REGION Network 6: Выходной сигнал контроллера
   RUNG wire#powerrail
      Contact( #CMD.Start_M )
      Move(in := 1, out1 => #Status)
      I_Contact( #Use.Inverse )
      wire#w1
      I_Contact( #All_Block )
      I_Contact( "Sim_All" )
      I_Contact( #CMD.Sim )
      I_Contact( #CMD.Local )
      Coil( #Q )
   END_RUNG
   RUNG wire#powerrail
      I_Contact( #CMD.Start_M )
      Move(in := 0, out1 => #Status)
      Contact( #Use.Inverse )
   END_RUNG wire#w1
   // the same network as SCL:
   IF #CMD.Start_M THEN #Status := 1; END_IF;
   IF NOT #CMD.Start_M THEN #Status := 0; END_IF;
   #Q := ((#CMD.Start_M AND NOT #Use.Inverse) OR (NOT #CMD.Start_M AND #Use.Inverse)) AND NOT #All_Block AND NOT "Sim_All" AND NOT #CMD.Sim AND NOT #CMD.Local;
END_REGION

REGION Network 7: Косвенная адресация
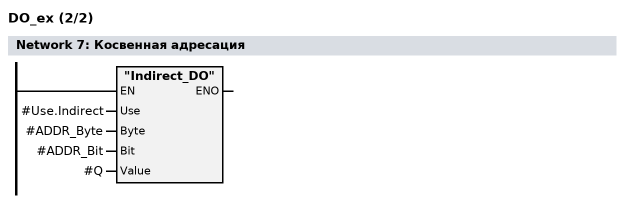
   RUNG wire#powerrail
      "Indirect_DO"(Use := #Use.Indirect, "Byte" := #ADDR_Byte, Bit := #ADDR_Bit, Value := #Q)
   END_RUNG
   // the same network as SCL:
   "Indirect_DO"(Use := #Use.Indirect, "Byte" := #ADDR_Byte, Bit := #ADDR_Bit, Value := #Q);
END_REGION
END_FUNCTION_BLOCK

FUNCTION_BLOCK "Motors"   // FB240, LAD
{ S7_Optimized_Access := 'FALSE' }
VERSION : 0.1
// stored: AutoNumber false, IsIECCheckEnabled false, SetENOAutomatically false, UDAEnableTagReadback false
   VAR DB_SPECIFIC
      Time_DTL { S7_SetPoint := 'True'} : DTL;
   END_VAR
BEGIN

REGION Network 1: Мешалки
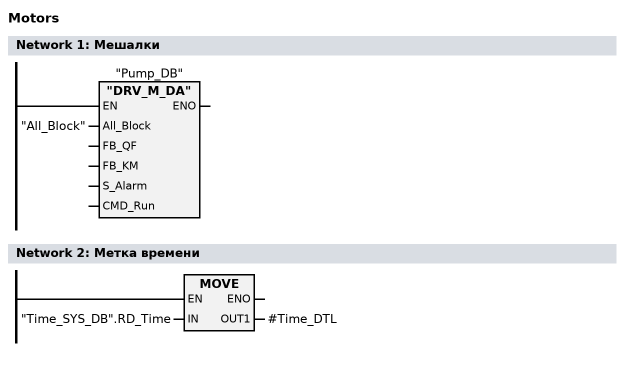
   RUNG wire#powerrail
      "Pump_DB"(All_Block := "All_Block", FB_QF :=, FB_KM :=, S_Alarm :=, CMD_Run :=)
   END_RUNG
   // the same network as SCL:
   "Pump_DB"(All_Block := "All_Block");   // "DRV_M_DA"
END_REGION

REGION Network 2: Метка времени
   RUNG wire#powerrail
      Move(in := "Time_SYS_DB".RD_Time, out1 => #Time_DTL)
   END_RUNG
   // the same network as SCL:
   #Time_DTL := "Time_SYS_DB".RD_Time;
END_REGION
END_FUNCTION_BLOCK

FUNCTION_BLOCK "DRV_M_DA"   // FB111, LAD
{ S7_Optimized_Access := 'FALSE' }
VERSION : 0.1
// stored: AutoNumber false, IsIECCheckEnabled false, SetENOAutomatically false, UDAEnableTagReadback false
   VAR_INPUT
      All_Block : Bool;   // Аварийный останов
   END_VAR
   VAR_IN_OUT
      FB_QF : Bool;   // защитный автомат / Защитный автомат / Готовность
      FB_KM : Bool;   // привод запущен / Пускатель / В работе
      S_Alarm : Bool;   // Внешний индикатор наличия аварии
      CMD_Run : Bool;   // Команда запуска двигателя
   END_VAR
   VAR DB_SPECIFIC
      CMD : "CMD";   // Основные команды / Блок команд
      Mode : Int;   // Режим работы
      Status : Int;   // Статус устройства
      Use : Struct   // Функционал
         QF { S7_SetPoint := 'True'} : Bool := true;   // Защитный автомат
         KM { S7_SetPoint := 'True'} : Bool := true;   // Пускатель
         OpTime { S7_SetPoint := 'True'} : Bool := true;   // Контроль наработки
         Analog { S7_SetPoint := 'True'} : Bool := true;
         Local_Keys : Bool;
      END_STRUCT;
      FB : Struct   // Функционал
         QF : Bool;   // Защитный автомат
         KM : Bool;   // Пускатель
         Local_Start : Bool;
         Local_Stop : Bool;
      END_STRUCT;
      ON : Bool;   // Успешно запущено
      OFF : Bool;   // Успешно остановлено
   END_VAR
   VAR
      Tx { S7_SetPoint := 'True'} : Array[0..3] of "Time_S";   // Блок таймеров
   END_VAR
   VAR DB_SPECIFIC
      Inv : Struct   // Инверсия сигналов
         CMD { S7_SetPoint := 'True'} : Bool;   // Команда запуска
         QF { S7_SetPoint := 'True'} : Bool;   // Защитный автомат
         KM { S7_SetPoint := 'True'} : Bool;   // Пускатель
      END_STRUCT;
      Alarm : Struct   // Сбор аварий / Список аварий
         Block : Bool;   // Аварийная остановка
         QF : Bool;   // привод не готов / Выбило защитный автомат
         Start : Bool;   // Ошибка при запуске
         Stop : Bool;   // Ошибка при останове
         Termo : Bool;   // термозащита / Сработала термозащита
         Alarm : Bool;   // Внешняя авария
         Safety : Bool;   // Сработала безопасность
         OpTime : Bool;
      END_STRUCT;
      Alarms : Word;   // Слово аварий
      Events : Word;   // События
      pos : Array[0..15] of Bool;
      OpTime_h : DInt;   // наработка (ч)
      OpTime_s { S7_SetPoint := 'True'} : DInt;   // наработка (с)
      OpTime_SP { S7_SetPoint := 'True'} : DInt := 2160;   // Интервал обслуживания, ч
      OpTime_Now_h : DInt;   // Прошло с прошлого обслуживания, ч
      OpTime_Now_s { S7_SetPoint := 'True'} : DInt;   // Прошло с прошлого обслуживания, с
      CodeID { S7_SetPoint := 'True'} : Int;   // Код датчика для привязки в скаде
      Indirect : Struct   // Использование косвенной адресации
         FB_QF { S7_SetPoint := 'True'} : Bool := true;   // защитный автомат / Защитный автомат
         FB_KM { S7_SetPoint := 'True'} : Bool := true;   // привод запущен / Пускатель
         CMD { S7_SetPoint := 'True'} : Bool := true;   // Команда запуска привода
      END_STRUCT;
      Indirect_BYTE : Struct   // Адрес входа на контроллере (Байт)
         FB_QF { S7_SetPoint := 'True'} : Int;   // защитный автомат / Защитный автомат
         FB_KM { S7_SetPoint := 'True'} : Int;   // привод запущен / Пускатель
         CMD { S7_SetPoint := 'True'} : Int;   // Команда запуска привода
      END_STRUCT;
      Indirect_BIT : Struct   // Адрес входа на контроллере (Бит)
         FB_QF { S7_SetPoint := 'True'} : Int := 9;   // защитный автомат / Защитный автомат
         FB_KM { S7_SetPoint := 'True'} : Int := 9;   // привод запущен / Пускатель
         CMD { S7_SetPoint := 'True'} : Int := 9;   // Команда запуска привода
      END_STRUCT;
      SP_A : Real;   // Уставка скорости в авторежиме
      SP_M : Real;   // Уставка скорости в ручном режиме
      ADDR { S7_SetPoint := 'True'} : Int;   // Уставка
   END_VAR
   VAR
      Converter { S7_SetPoint := 'True'} : "Converter_SCL";   // Масштабирование сигнала
   END_VAR
   VAR DB_SPECIFIC
      VmA : Real;   // Реальный сигнал на входе ПЛК
      Output_Type { S7_SetPoint := 'True'} : Int;   // Тип выхода, 0 - 4..20, 1 - 0..20, 2 - 0..10, 3 - 0..5
      "Type" { S7_SetPoint := 'True'} : Int;   // Размерность
   END_VAR
   VAR
      Slow { S7_SetPoint := 'True'} : "Slow";   // Плавный разгон и замедление
   END_VAR
   VAR DB_SPECIFIC
      "Name" { S7_SetPoint := 'True'} : String[4];
      coeff : Real;
      SP_Min { S7_SetPoint := 'True'} : Real := 30.0;
      Time_DTL { S7_SetPoint := 'True'} : DTL;
   END_VAR
   VAR_TEMP
      ev : Bool;
      xQF : Bool;
      xKM : Bool;
      xSP : Real;
      Signal_R : Real;   // Актуальный сигнал
      Signal_Dint : DInt;   // Сигнал в DInt
      Signal_Ex : Int;   // Конвертация сигнала
      Type_Min : Real;
      Type_Max : Real;
   END_VAR
   // Converter.Max_In := 100.0;
   // Converter.Max_Out := 27648.0;
   VAR_TEMP   // added for the SCL form of the ladder/FBD networks
      _w1 : Bool;
      _w2 : Bool;
      _w3 : Bool;
      _w4 : Bool;
      _w5 : Bool;
      _w6 : Bool;
      _w7 : Bool;
      _w8 : Bool;
      _w9 : Bool;
      _w10 : Bool;
      _w11 : Bool;
      _w12 : Bool;
      _w13 : Bool;
      _w14 : Bool;
      _w15 : Bool;
      _w16 : Bool;
      _w17 : Bool;
      _w18 : Bool;
      _w19 : Bool;
      _w20 : Bool;
      _w21 : Bool;
      _w22 : Bool;
      _w23 : Bool;
      _w24 : Bool;
      _w25 : Bool;
      _w26 : Bool;
   END_VAR
BEGIN

REGION Network 1: Режим глобальной симуляции
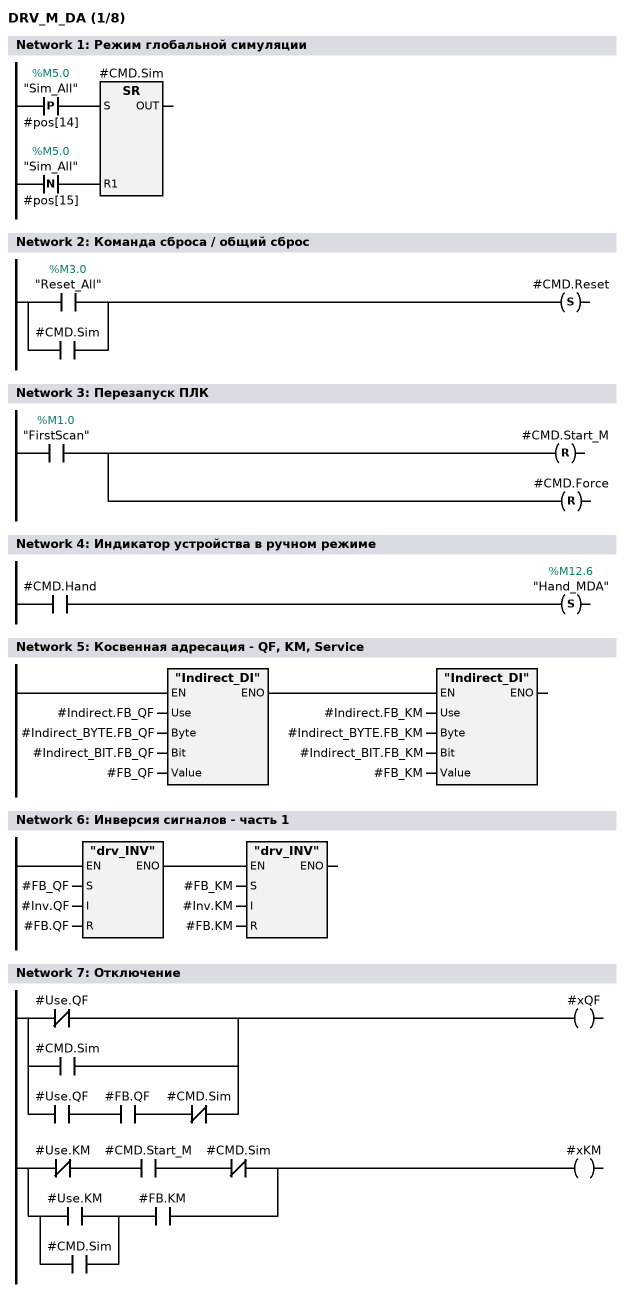
   RUNG wire#powerrail
      P_Contact(operand := "Sim_All", bit := #pos[14])
      S_SR(operand := #CMD.Sim, r1 := wire#w1)
   END_RUNG
   RUNG wire#powerrail
      N_Contact(operand := "Sim_All", bit := #pos[15])
   END_RUNG wire#w1
   // the same network as SCL:
   #_w1 := "Sim_All" AND NOT #pos[14];   // rising edge of "Sim_All"
   #pos[14] := "Sim_All";
   #_w2 := NOT "Sim_All" AND #pos[15];   // falling edge of "Sim_All"
   #pos[15] := "Sim_All";
   IF #_w1 THEN
       #CMD.Sim := TRUE;   // SR flip-flop
   END_IF;
   IF #_w2 THEN #CMD.Sim := FALSE; END_IF;
END_REGION

REGION Network 2: Команда сброса / общий сброс
   RUNG wire#powerrail
      Contact( "Reset_All" )
      wire#w1
      S_Coil( #CMD.Reset )
   END_RUNG
   RUNG wire#powerrail
      Contact( #CMD.Sim )
   END_RUNG wire#w1
   // the same network as SCL:
   IF "Reset_All" OR #CMD.Sim THEN #CMD.Reset := TRUE; END_IF;
END_REGION

REGION Network 3: Перезапуск ПЛК
   RUNG wire#powerrail
      Contact( "FirstScan" )
      wire#w1
      R_Coil( #CMD.Start_M )
   END_RUNG
   RUNG wire#w1
      R_Coil( #CMD.Force )
   END_RUNG
   // the same network as SCL:
   IF "FirstScan" THEN
       #CMD.Start_M := FALSE;
       #CMD.Force := FALSE;
   END_IF;
END_REGION

REGION Network 4: Индикатор устройства в ручном режиме
   RUNG wire#powerrail
      Contact( #CMD.Hand )
      S_Coil( "Hand_MDA" )
   END_RUNG
   // the same network as SCL:
   IF #CMD.Hand THEN "Hand_MDA" := TRUE; END_IF;
END_REGION

REGION Network 5: Косвенная адресация - QF, KM, Service
   RUNG wire#powerrail
      "Indirect_DI"(Use := #Indirect.FB_QF, "Byte" := #Indirect_BYTE.FB_QF, Bit := #Indirect_BIT.FB_QF, Value := #FB_QF)
      "Indirect_DI"(Use := #Indirect.FB_KM, "Byte" := #Indirect_BYTE.FB_KM, Bit := #Indirect_BIT.FB_KM, Value := #FB_KM)
   END_RUNG
   // the same network as SCL:
   "Indirect_DI"(Use := #Indirect.FB_QF,
                 "Byte" := #Indirect_BYTE.FB_QF,
                 Bit := #Indirect_BIT.FB_QF,
                 Value := #FB_QF,
                 ENO => #_w1);
   IF #_w1 THEN
       "Indirect_DI"(Use := #Indirect.FB_KM,
                     "Byte" := #Indirect_BYTE.FB_KM,
                     Bit := #Indirect_BIT.FB_KM,
                     Value := #FB_KM);
   END_IF;
END_REGION

REGION Network 6: Инверсия сигналов - часть 1
   RUNG wire#powerrail
      "drv_INV"(S := #FB_QF, I := #Inv.QF, R := #FB.QF)
      "drv_INV"(S := #FB_KM, I := #Inv.KM, R := #FB.KM)
   END_RUNG
   // the same network as SCL:
   "drv_INV"(S := #FB_QF, I := #Inv.QF, R := #FB.QF, ENO => #_w1);
   IF #_w1 THEN "drv_INV"(S := #FB_KM, I := #Inv.KM, R := #FB.KM); END_IF;
END_REGION

REGION Network 7: Отключение
   RUNG wire#powerrail
      I_Contact( #Use.QF )
      wire#w1
      Coil( #xQF )
   END_RUNG
   RUNG wire#powerrail
      Contact( #CMD.Sim )
   END_RUNG wire#w1
   RUNG wire#powerrail
      Contact( #Use.QF )
      Contact( #FB.QF )
      I_Contact( #CMD.Sim )
   END_RUNG wire#w1
   RUNG wire#powerrail
      I_Contact( #Use.KM )
      Contact( #CMD.Start_M )
      I_Contact( #CMD.Sim )
      wire#w2
      Coil( #xKM )
   END_RUNG
   RUNG wire#powerrail
      Contact( #Use.KM )
      wire#w3
      Contact( #FB.KM )
   END_RUNG wire#w2
   RUNG wire#powerrail
      Contact( #CMD.Sim )
   END_RUNG wire#w3
   // the same network as SCL:
   #xQF := NOT #Use.QF OR #CMD.Sim OR (#Use.QF AND #FB.QF AND NOT #CMD.Sim);
   #xKM := (NOT #Use.KM AND #CMD.Start_M AND NOT #CMD.Sim) OR ((#Use.KM OR #CMD.Sim) AND #FB.KM);
END_REGION

REGION Network 8: Режим работы устройства / определение режима работы
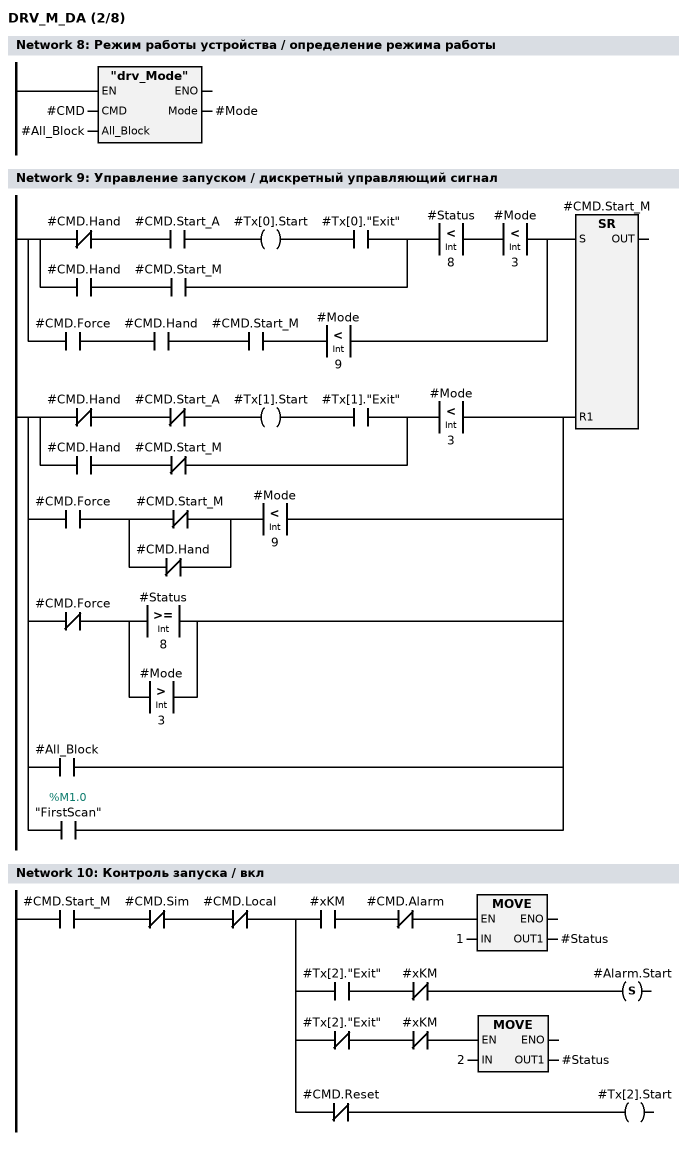
   RUNG wire#powerrail
      "drv_Mode"(CMD := #CMD, All_Block := #All_Block, Mode => #Mode)
   END_RUNG
   // the same network as SCL:
   "drv_Mode"(CMD := #CMD, All_Block := #All_Block, Mode => #Mode);
END_REGION

REGION Network 9: Управление запуском / дискретный управляющий сигнал
   RUNG wire#powerrail
      I_Contact( #CMD.Hand )
      Contact( #CMD.Start_A )
      Coil( #Tx[0].Start )
      Contact( #Tx[0]."Exit" )
      wire#w1
      { S7_Templates := "SrcType := Int" } LT_Contact(in1 := #Status, in2 := 8)
      { S7_Templates := "SrcType := Int" } LT_Contact(in1 := #Mode, in2 := 3)
      wire#w2
      S_SR(operand := #CMD.Start_M, r1 := wire#w7)
   END_RUNG
   RUNG wire#powerrail
      Contact( #CMD.Hand )
      Contact( #CMD.Start_M )
   END_RUNG wire#w1
   RUNG wire#powerrail
      Contact( #CMD.Force )
      Contact( #CMD.Hand )
      Contact( #CMD.Start_M )
      { S7_Templates := "SrcType := Int" } LT_Contact(in1 := #Mode, in2 := 9)
   END_RUNG wire#w2
   RUNG wire#powerrail
      I_Contact( #CMD.Hand )
      I_Contact( #CMD.Start_A )
      Coil( #Tx[1].Start )
      Contact( #Tx[1]."Exit" )
      wire#w3
      { S7_Templates := "SrcType := Int" } LT_Contact(in1 := #Mode, in2 := 3)
   END_RUNG wire#w7
   RUNG wire#powerrail
      Contact( #CMD.Hand )
      I_Contact( #CMD.Start_M )
   END_RUNG wire#w3
   RUNG wire#powerrail
      Contact( #CMD.Force )
      wire#w4
      I_Contact( #CMD.Start_M )
      wire#w5
      { S7_Templates := "SrcType := Int" } LT_Contact(in1 := #Mode, in2 := 9)
   END_RUNG wire#w7
   RUNG wire#w4
      I_Contact( #CMD.Hand )
   END_RUNG wire#w5
   RUNG wire#powerrail
      I_Contact( #CMD.Force )
      wire#w6
      { S7_Templates := "SrcType := Int" } GE_Contact(in1 := #Status, in2 := 8)
   END_RUNG wire#w7
   RUNG wire#w6
      { S7_Templates := "SrcType := Int" } GT_Contact(in1 := #Mode, in2 := 3)
   END_RUNG wire#w7
   RUNG wire#powerrail
      Contact( #All_Block )
   END_RUNG wire#w7
   RUNG wire#powerrail
      Contact( "FirstScan" )
   END_RUNG wire#w7
   // the same network as SCL:
   #Tx[0].Start := NOT #CMD.Hand AND #CMD.Start_A;
   #_w1 := (((NOT #CMD.Hand AND #CMD.Start_A AND #Tx[0]."Exit") OR (#CMD.Hand AND #CMD.Start_M)) AND (#Status < 8) AND (#Mode < 3)) OR (#CMD.Force AND #CMD.Hand AND #CMD.Start_M AND (#Mode < 9));
   #Tx[1].Start := NOT #CMD.Hand AND NOT #CMD.Start_A;
   #_w2 := (((NOT #CMD.Hand AND NOT #CMD.Start_A AND #Tx[1]."Exit") OR (#CMD.Hand AND NOT #CMD.Start_M)) AND (#Mode < 3)) OR (#CMD.Force AND (NOT #CMD.Start_M OR NOT #CMD.Hand) AND (#Mode < 9)) OR (NOT #CMD.Force AND ((#Status >= 8) OR (#Mode > 3))) OR #All_Block OR "FirstScan";
   IF #_w1 THEN
       #CMD.Start_M := TRUE;   // SR flip-flop
   END_IF;
   IF #_w2 THEN #CMD.Start_M := FALSE; END_IF;
END_REGION

REGION Network 10: Контроль запуска / вкл
   RUNG wire#powerrail
      Contact( #CMD.Start_M )
      I_Contact( #CMD.Sim )
      I_Contact( #CMD.Local )
      wire#w1
      Contact( #xKM )
      I_Contact( #CMD.Alarm )
      { S7_GenerateENO := "TRUE" } Move(in := 1, out1 => #Status)
   END_RUNG
   RUNG wire#w1
      Contact( #Tx[2]."Exit" )
      I_Contact( #xKM )
      S_Coil( #Alarm.Start )
   END_RUNG
   RUNG wire#w1
      I_Contact( #Tx[2]."Exit" )
      I_Contact( #xKM )
      { S7_GenerateENO := "TRUE" } Move(in := 2, out1 => #Status)
   END_RUNG
   RUNG wire#w1
      I_Contact( #CMD.Reset )
      Coil( #Tx[2].Start )
   END_RUNG
   // the same network as SCL:
   #_w1 := #CMD.Start_M AND NOT #CMD.Sim AND NOT #CMD.Local;
   IF #_w1 AND #xKM AND NOT #CMD.Alarm THEN #Status := 1; END_IF;
   IF #_w1 AND #Tx[2]."Exit" AND NOT #xKM THEN #Alarm.Start := TRUE; END_IF;
   IF #_w1 AND NOT #Tx[2]."Exit" AND NOT #xKM THEN #Status := 2; END_IF;
   #Tx[2].Start := #_w1 AND NOT #CMD.Reset;
END_REGION

REGION Network 11: Контроль останова / выкл
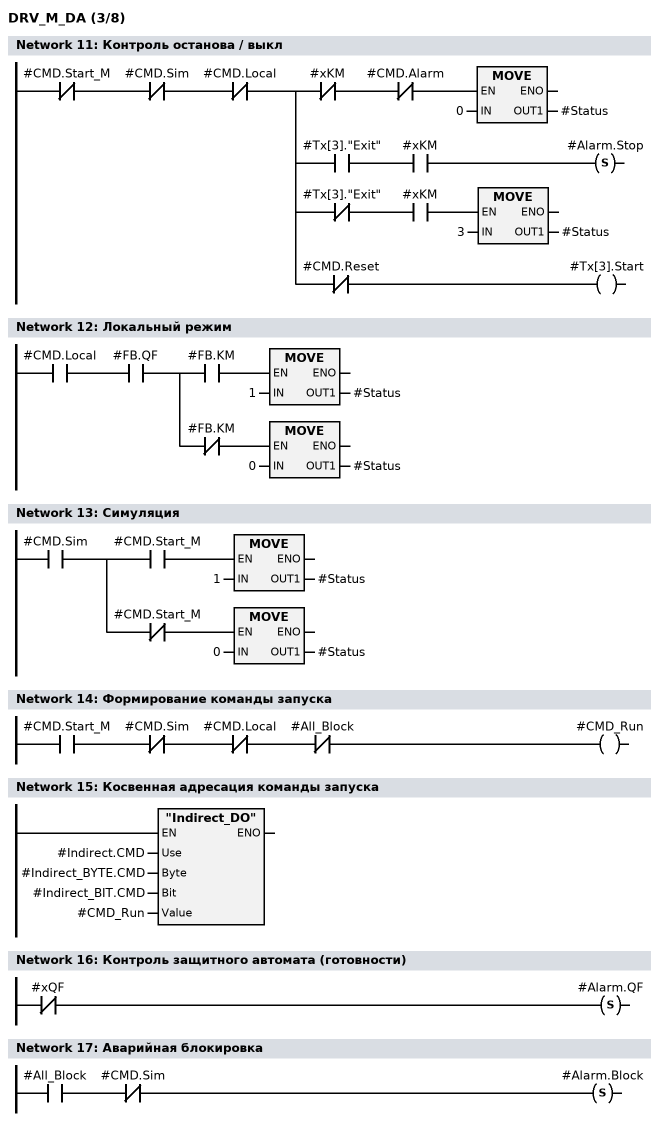
   RUNG wire#powerrail
      I_Contact( #CMD.Start_M )
      I_Contact( #CMD.Sim )
      I_Contact( #CMD.Local )
      wire#w1
      I_Contact( #xKM )
      I_Contact( #CMD.Alarm )
      { S7_GenerateENO := "TRUE" } Move(in := 0, out1 => #Status)
   END_RUNG
   RUNG wire#w1
      Contact( #Tx[3]."Exit" )
      Contact( #xKM )
      S_Coil( #Alarm.Stop )
   END_RUNG
   RUNG wire#w1
      I_Contact( #Tx[3]."Exit" )
      Contact( #xKM )
      { S7_GenerateENO := "TRUE" } Move(in := 3, out1 => #Status)
   END_RUNG
   RUNG wire#w1
      I_Contact( #CMD.Reset )
      Coil( #Tx[3].Start )
   END_RUNG
   // the same network as SCL:
   #_w1 := NOT #CMD.Start_M AND NOT #CMD.Sim AND NOT #CMD.Local;
   IF #_w1 AND NOT #xKM AND NOT #CMD.Alarm THEN #Status := 0; END_IF;
   IF #_w1 AND #Tx[3]."Exit" AND #xKM THEN #Alarm.Stop := TRUE; END_IF;
   IF #_w1 AND NOT #Tx[3]."Exit" AND #xKM THEN #Status := 3; END_IF;
   #Tx[3].Start := #_w1 AND NOT #CMD.Reset;
END_REGION

REGION Network 12: Локальный режим
   RUNG wire#powerrail
      Contact( #CMD.Local )
      Contact( #FB.QF )
      wire#w1
      Contact( #FB.KM )
      { S7_GenerateENO := "TRUE" } Move(in := 1, out1 => #Status)
   END_RUNG
   RUNG wire#w1
      I_Contact( #FB.KM )
      { S7_GenerateENO := "TRUE" } Move(in := 0, out1 => #Status)
   END_RUNG
   // the same network as SCL:
   #_w1 := #CMD.Local AND #FB.QF;
   IF #_w1 AND #FB.KM THEN #Status := 1; END_IF;
   IF #_w1 AND NOT #FB.KM THEN #Status := 0; END_IF;
END_REGION

REGION Network 13: Симуляция
   RUNG wire#powerrail
      Contact( #CMD.Sim )
      wire#w1
      Contact( #CMD.Start_M )
      { S7_GenerateENO := "TRUE" } Move(in := 1, out1 => #Status)
   END_RUNG
   RUNG wire#w1
      I_Contact( #CMD.Start_M )
      { S7_GenerateENO := "TRUE" } Move(in := 0, out1 => #Status)
   END_RUNG
   // the same network as SCL:
   IF #CMD.Sim AND #CMD.Start_M THEN #Status := 1; END_IF;
   IF #CMD.Sim AND NOT #CMD.Start_M THEN #Status := 0; END_IF;
END_REGION

REGION Network 14: Формирование команды запуска
   RUNG wire#powerrail
      Contact( #CMD.Start_M )
      I_Contact( #CMD.Sim )
      I_Contact( #CMD.Local )
      I_Contact( #All_Block )
      Coil( #CMD_Run )
   END_RUNG
   // the same network as SCL:
   #CMD_Run := #CMD.Start_M AND NOT #CMD.Sim AND NOT #CMD.Local AND NOT #All_Block;
END_REGION

REGION Network 15: Косвенная адресация команды запуска
   RUNG wire#powerrail
      "Indirect_DO"(Use := #Indirect.CMD, "Byte" := #Indirect_BYTE.CMD, Bit := #Indirect_BIT.CMD, Value := #CMD_Run)
   END_RUNG
   // the same network as SCL:
   "Indirect_DO"(Use := #Indirect.CMD,
                 "Byte" := #Indirect_BYTE.CMD,
                 Bit := #Indirect_BIT.CMD,
                 Value := #CMD_Run);
END_REGION

REGION Network 16: Контроль защитного автомата (готовности)
   RUNG wire#powerrail
      I_Contact( #xQF )
      S_Coil( #Alarm.QF )
   END_RUNG
   // the same network as SCL:
   IF NOT #xQF THEN #Alarm.QF := TRUE; END_IF;
END_REGION

REGION Network 17: Аварийная блокировка
   RUNG wire#powerrail
      Contact( #All_Block )
      I_Contact( #CMD.Sim )
      S_Coil( #Alarm.Block )
   END_RUNG
   // the same network as SCL:
   IF #All_Block AND NOT #CMD.Sim THEN #Alarm.Block := TRUE; END_IF;
END_REGION

REGION Network 18: Сигнал аварии
   // Safety - сработал датчик безопасности, подключается через отдельный дискретный вход
   // Termo - сработала термозащита, подключается через отдельный дискретный вход
   // Alarm - сработала внешняя авария, подключается через отдельный дискретный вход
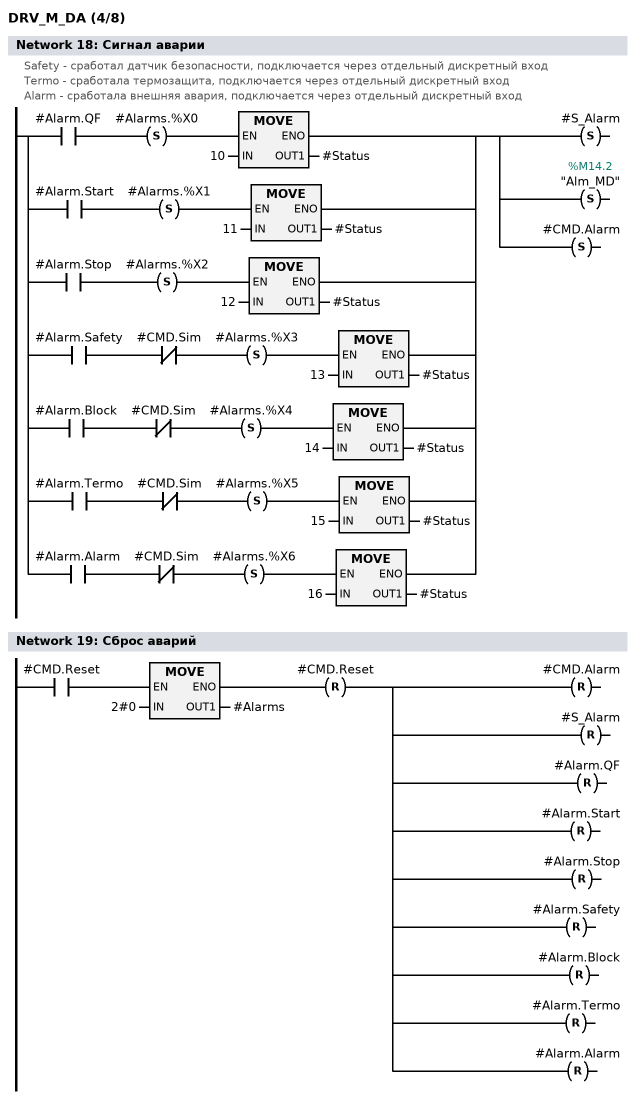
   RUNG wire#powerrail
      Contact( #Alarm.QF )
      S_Coil( #Alarms.%X0 )
      { S7_GenerateENO := "TRUE" } Move(in := 10, out1 => #Status)
      wire#w1
      S_Coil( #S_Alarm )
   END_RUNG
   RUNG wire#powerrail
      Contact( #Alarm.Start )
      S_Coil( #Alarms.%X1 )
      { S7_GenerateENO := "TRUE" } Move(in := 11, out1 => #Status)
   END_RUNG wire#w1
   RUNG wire#powerrail
      Contact( #Alarm.Stop )
      S_Coil( #Alarms.%X2 )
      { S7_GenerateENO := "TRUE" } Move(in := 12, out1 => #Status)
   END_RUNG wire#w1
   RUNG wire#powerrail
      Contact( #Alarm.Safety )
      I_Contact( #CMD.Sim )
      S_Coil( #Alarms.%X3 )
      { S7_GenerateENO := "TRUE" } Move(in := 13, out1 => #Status)
   END_RUNG wire#w1
   RUNG wire#powerrail
      Contact( #Alarm.Block )
      I_Contact( #CMD.Sim )
      S_Coil( #Alarms.%X4 )
      { S7_GenerateENO := "TRUE" } Move(in := 14, out1 => #Status)
   END_RUNG wire#w1
   RUNG wire#powerrail
      Contact( #Alarm.Termo )
      I_Contact( #CMD.Sim )
      S_Coil( #Alarms.%X5 )
      { S7_GenerateENO := "TRUE" } Move(in := 15, out1 => #Status)
   END_RUNG wire#w1
   RUNG wire#powerrail
      Contact( #Alarm.Alarm )
      I_Contact( #CMD.Sim )
      S_Coil( #Alarms.%X6 )
      { S7_GenerateENO := "TRUE" } Move(in := 16, out1 => #Status)
   END_RUNG wire#w1
   RUNG wire#w1
      S_Coil( "Alm_MD" )
   END_RUNG
   RUNG wire#w1
      S_Coil( #CMD.Alarm )
   END_RUNG
   // the same network as SCL:
   // ENO of a box is taken as its EN; it also drops when the box reports an error
   IF #Alarm.QF THEN
       #Alarms.%X0 := TRUE;
       #Status := 10;
   END_IF;
   IF #Alarm.Start THEN
       #Alarms.%X1 := TRUE;
       #Status := 11;
   END_IF;
   IF #Alarm.Stop THEN
       #Alarms.%X2 := TRUE;
       #Status := 12;
   END_IF;
   #_w1 := #Alarm.Safety AND NOT #CMD.Sim;
   IF #_w1 THEN
       #Alarms.%X3 := TRUE;
       #Status := 13;
   END_IF;
   #_w2 := #Alarm.Block AND NOT #CMD.Sim;
   IF #_w2 THEN
       #Alarms.%X4 := TRUE;
       #Status := 14;
   END_IF;
   #_w3 := #Alarm.Termo AND NOT #CMD.Sim;
   IF #_w3 THEN
       #Alarms.%X5 := TRUE;
       #Status := 15;
   END_IF;
   #_w4 := #Alarm.Alarm AND NOT #CMD.Sim;
   IF #_w4 THEN
       #Alarms.%X6 := TRUE;
       #Status := 16;
   END_IF;
   IF #Alarm.QF OR #Alarm.Start OR #Alarm.Stop OR #_w1 OR #_w2 OR #_w3 OR #_w4 THEN
       #S_Alarm := TRUE;
       "Alm_MD" := TRUE;
       #CMD.Alarm := TRUE;
   END_IF;
END_REGION

REGION Network 19: Сброс аварий
   RUNG wire#powerrail
      Contact( #CMD.Reset )
      Move(in := 2#0, out1 => #Alarms)
      R_Coil( #CMD.Reset )
      wire#w1
      R_Coil( #CMD.Alarm )
   END_RUNG
   RUNG wire#w1
      R_Coil( #S_Alarm )
   END_RUNG
   RUNG wire#w1
      R_Coil( #Alarm.QF )
   END_RUNG
   RUNG wire#w1
      R_Coil( #Alarm.Start )
   END_RUNG
   RUNG wire#w1
      R_Coil( #Alarm.Stop )
   END_RUNG
   RUNG wire#w1
      R_Coil( #Alarm.Safety )
   END_RUNG
   RUNG wire#w1
      R_Coil( #Alarm.Block )
   END_RUNG
   RUNG wire#w1
      R_Coil( #Alarm.Termo )
   END_RUNG
   RUNG wire#w1
      R_Coil( #Alarm.Alarm )
   END_RUNG
   // the same network as SCL:
   IF #CMD.Reset THEN #Alarms := 2#0; END_IF;
   #_w1 := #CMD.Reset;
   IF #_w1 THEN
       #CMD.Reset := FALSE;
       #CMD.Alarm := FALSE;
       #S_Alarm := FALSE;
       #Alarm.QF := FALSE;
       #Alarm.Start := FALSE;
       #Alarm.Stop := FALSE;
       #Alarm.Safety := FALSE;
       #Alarm.Block := FALSE;
       #Alarm.Termo := FALSE;
       #Alarm.Alarm := FALSE;
   END_IF;
END_REGION

REGION Network 20: События привода
   // 0 - ручной режим активирован
   // 1 - ручной режим деактивирован
   // 2 - принудительный режим активирован
   // 3 - принудительный режим деактивирован
   // 4 - запуск в ручном режиме
   // 5 - останов в ручном режиме
   // 6 - местный режим управления активирован
   // 7 - местный режим управления деактивирован
   // 8 - запущено в местном режиме
   // 9 - остановлено в местном режиме
   // 10 - сервисный режим активирован
   // 11 - сервисный режим деактивирован
   // 12 - проведено сервисное обслуживание
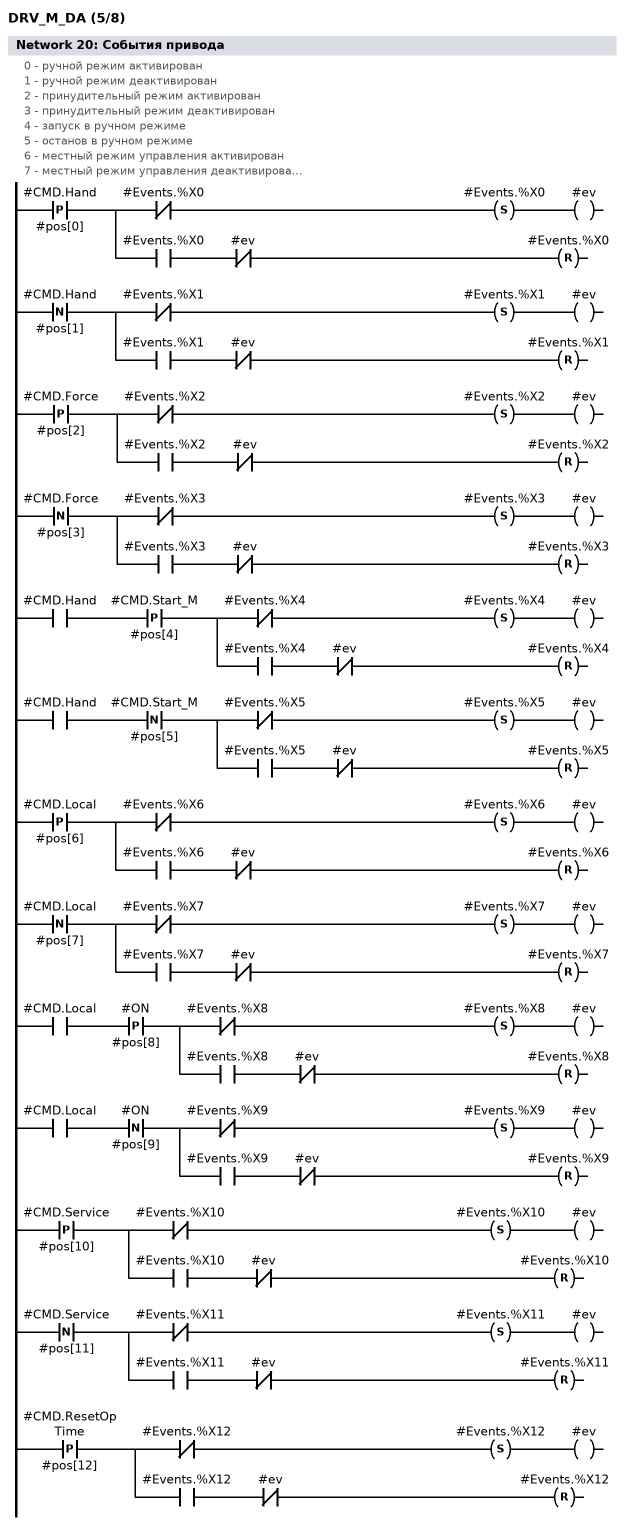
   RUNG wire#powerrail
      P_Contact(operand := #CMD.Hand, bit := #pos[0])
      wire#w1
      I_Contact( #Events.%X0 )
      S_Coil( #Events.%X0 )
      Coil( #ev )
   END_RUNG
   RUNG wire#w1
      Contact( #Events.%X0 )
      I_Contact( #ev )
      R_Coil( #Events.%X0 )
   END_RUNG
   RUNG wire#powerrail
      N_Contact(operand := #CMD.Hand, bit := #pos[1])
      wire#w2
      I_Contact( #Events.%X1 )
      S_Coil( #Events.%X1 )
      Coil( #ev )
   END_RUNG
   RUNG wire#w2
      Contact( #Events.%X1 )
      I_Contact( #ev )
      R_Coil( #Events.%X1 )
   END_RUNG
   RUNG wire#powerrail
      P_Contact(operand := #CMD.Force, bit := #pos[2])
      wire#w3
      I_Contact( #Events.%X2 )
      S_Coil( #Events.%X2 )
      Coil( #ev )
   END_RUNG
   RUNG wire#w3
      Contact( #Events.%X2 )
      I_Contact( #ev )
      R_Coil( #Events.%X2 )
   END_RUNG
   RUNG wire#powerrail
      N_Contact(operand := #CMD.Force, bit := #pos[3])
      wire#w4
      I_Contact( #Events.%X3 )
      S_Coil( #Events.%X3 )
      Coil( #ev )
   END_RUNG
   RUNG wire#w4
      Contact( #Events.%X3 )
      I_Contact( #ev )
      R_Coil( #Events.%X3 )
   END_RUNG
   RUNG wire#powerrail
      Contact( #CMD.Hand )
      P_Contact(operand := #CMD.Start_M, bit := #pos[4])
      wire#w5
      I_Contact( #Events.%X4 )
      S_Coil( #Events.%X4 )
      Coil( #ev )
   END_RUNG
   RUNG wire#w5
      Contact( #Events.%X4 )
      I_Contact( #ev )
      R_Coil( #Events.%X4 )
   END_RUNG
   RUNG wire#powerrail
      Contact( #CMD.Hand )
      N_Contact(operand := #CMD.Start_M, bit := #pos[5])
      wire#w6
      I_Contact( #Events.%X5 )
      S_Coil( #Events.%X5 )
      Coil( #ev )
   END_RUNG
   RUNG wire#w6
      Contact( #Events.%X5 )
      I_Contact( #ev )
      R_Coil( #Events.%X5 )
   END_RUNG
   RUNG wire#powerrail
      P_Contact(operand := #CMD.Local, bit := #pos[6])
      wire#w7
      I_Contact( #Events.%X6 )
      S_Coil( #Events.%X6 )
      Coil( #ev )
   END_RUNG
   RUNG wire#w7
      Contact( #Events.%X6 )
      I_Contact( #ev )
      R_Coil( #Events.%X6 )
   END_RUNG
   RUNG wire#powerrail
      N_Contact(operand := #CMD.Local, bit := #pos[7])
      wire#w8
      I_Contact( #Events.%X7 )
      S_Coil( #Events.%X7 )
      Coil( #ev )
   END_RUNG
   RUNG wire#w8
      Contact( #Events.%X7 )
      I_Contact( #ev )
      R_Coil( #Events.%X7 )
   END_RUNG
   RUNG wire#powerrail
      Contact( #CMD.Local )
      P_Contact(operand := #ON, bit := #pos[8])
      wire#w9
      I_Contact( #Events.%X8 )
      S_Coil( #Events.%X8 )
      Coil( #ev )
   END_RUNG
   RUNG wire#w9
      Contact( #Events.%X8 )
      I_Contact( #ev )
      R_Coil( #Events.%X8 )
   END_RUNG
   RUNG wire#powerrail
      Contact( #CMD.Local )
      N_Contact(operand := #ON, bit := #pos[9])
      wire#w10
      I_Contact( #Events.%X9 )
      S_Coil( #Events.%X9 )
      Coil( #ev )
   END_RUNG
   RUNG wire#w10
      Contact( #Events.%X9 )
      I_Contact( #ev )
      R_Coil( #Events.%X9 )
   END_RUNG
   RUNG wire#powerrail
      P_Contact(operand := #CMD.Service, bit := #pos[10])
      wire#w11
      I_Contact( #Events.%X10 )
      S_Coil( #Events.%X10 )
      Coil( #ev )
   END_RUNG
   RUNG wire#w11
      Contact( #Events.%X10 )
      I_Contact( #ev )
      R_Coil( #Events.%X10 )
   END_RUNG
   RUNG wire#powerrail
      N_Contact(operand := #CMD.Service, bit := #pos[11])
      wire#w12
      I_Contact( #Events.%X11 )
      S_Coil( #Events.%X11 )
      Coil( #ev )
   END_RUNG
   RUNG wire#w12
      Contact( #Events.%X11 )
      I_Contact( #ev )
      R_Coil( #Events.%X11 )
   END_RUNG
   RUNG wire#powerrail
      P_Contact(operand := #CMD.ResetOpTime, bit := #pos[12])
      wire#w13
      I_Contact( #Events.%X12 )
      S_Coil( #Events.%X12 )
      Coil( #ev )
   END_RUNG
   RUNG wire#w13
      Contact( #Events.%X12 )
      I_Contact( #ev )
      R_Coil( #Events.%X12 )
   END_RUNG
   // the same network as SCL:
   #_w1 := #CMD.Hand AND NOT #pos[0];   // rising edge of #CMD.Hand
   #pos[0] := #CMD.Hand;
   #_w2 := #_w1 AND NOT #Events.%X0;
   IF #_w2 THEN #Events.%X0 := TRUE; END_IF;
   #ev := #_w2;
   IF #_w1 AND #Events.%X0 AND NOT #ev THEN #Events.%X0 := FALSE; END_IF;
   #_w3 := NOT #CMD.Hand AND #pos[1];   // falling edge of #CMD.Hand
   #pos[1] := #CMD.Hand;
   #_w4 := #_w3 AND NOT #Events.%X1;
   IF #_w4 THEN #Events.%X1 := TRUE; END_IF;
   #ev := #_w4;
   IF #_w3 AND #Events.%X1 AND NOT #ev THEN #Events.%X1 := FALSE; END_IF;
   #_w5 := #CMD.Force AND NOT #pos[2];   // rising edge of #CMD.Force
   #pos[2] := #CMD.Force;
   #_w6 := #_w5 AND NOT #Events.%X2;
   IF #_w6 THEN #Events.%X2 := TRUE; END_IF;
   #ev := #_w6;
   IF #_w5 AND #Events.%X2 AND NOT #ev THEN #Events.%X2 := FALSE; END_IF;
   #_w7 := NOT #CMD.Force AND #pos[3];   // falling edge of #CMD.Force
   #pos[3] := #CMD.Force;
   #_w8 := #_w7 AND NOT #Events.%X3;
   IF #_w8 THEN #Events.%X3 := TRUE; END_IF;
   #ev := #_w8;
   IF #_w7 AND #Events.%X3 AND NOT #ev THEN #Events.%X3 := FALSE; END_IF;
   #_w9 := #CMD.Hand AND #CMD.Start_M AND NOT #pos[4];   // rising edge of #CMD.Start_M
   #pos[4] := #CMD.Start_M;
   #_w10 := #_w9 AND NOT #Events.%X4;
   IF #_w10 THEN #Events.%X4 := TRUE; END_IF;
   #ev := #_w10;
   IF #_w9 AND #Events.%X4 AND NOT #ev THEN #Events.%X4 := FALSE; END_IF;
   #_w11 := #CMD.Hand AND NOT #CMD.Start_M AND #pos[5];   // falling edge of #CMD.Start_M
   #pos[5] := #CMD.Start_M;
   #_w12 := #_w11 AND NOT #Events.%X5;
   IF #_w12 THEN #Events.%X5 := TRUE; END_IF;
   #ev := #_w12;
   IF #_w11 AND #Events.%X5 AND NOT #ev THEN #Events.%X5 := FALSE; END_IF;
   #_w13 := #CMD.Local AND NOT #pos[6];   // rising edge of #CMD.Local
   #pos[6] := #CMD.Local;
   #_w14 := #_w13 AND NOT #Events.%X6;
   IF #_w14 THEN #Events.%X6 := TRUE; END_IF;
   #ev := #_w14;
   IF #_w13 AND #Events.%X6 AND NOT #ev THEN #Events.%X6 := FALSE; END_IF;
   #_w15 := NOT #CMD.Local AND #pos[7];   // falling edge of #CMD.Local
   #pos[7] := #CMD.Local;
   #_w16 := #_w15 AND NOT #Events.%X7;
   IF #_w16 THEN #Events.%X7 := TRUE; END_IF;
   #ev := #_w16;
   IF #_w15 AND #Events.%X7 AND NOT #ev THEN #Events.%X7 := FALSE; END_IF;
   #_w17 := #CMD.Local AND #ON AND NOT #pos[8];   // rising edge of #ON
   #pos[8] := #ON;
   #_w18 := #_w17 AND NOT #Events.%X8;
   IF #_w18 THEN #Events.%X8 := TRUE; END_IF;
   #ev := #_w18;
   IF #_w17 AND #Events.%X8 AND NOT #ev THEN #Events.%X8 := FALSE; END_IF;
   #_w19 := #CMD.Local AND NOT #ON AND #pos[9];   // falling edge of #ON
   #pos[9] := #ON;
   #_w20 := #_w19 AND NOT #Events.%X9;
   IF #_w20 THEN #Events.%X9 := TRUE; END_IF;
   #ev := #_w20;
   IF #_w19 AND #Events.%X9 AND NOT #ev THEN #Events.%X9 := FALSE; END_IF;
   #_w21 := #CMD.Service AND NOT #pos[10];   // rising edge of #CMD.Service
   #pos[10] := #CMD.Service;
   #_w22 := #_w21 AND NOT #Events.%X10;
   IF #_w22 THEN #Events.%X10 := TRUE; END_IF;
   #ev := #_w22;
   IF #_w21 AND #Events.%X10 AND NOT #ev THEN #Events.%X10 := FALSE; END_IF;
   #_w23 := NOT #CMD.Service AND #pos[11];   // falling edge of #CMD.Service
   #pos[11] := #CMD.Service;
   #_w24 := #_w23 AND NOT #Events.%X11;
   IF #_w24 THEN #Events.%X11 := TRUE; END_IF;
   #ev := #_w24;
   IF #_w23 AND #Events.%X11 AND NOT #ev THEN #Events.%X11 := FALSE; END_IF;
   #_w25 := #CMD.ResetOpTime AND NOT #pos[12];   // rising edge of #CMD.ResetOpTime
   #pos[12] := #CMD.ResetOpTime;
   #_w26 := #_w25 AND NOT #Events.%X12;
   IF #_w26 THEN #Events.%X12 := TRUE; END_IF;
   #ev := #_w26;
   IF #_w25 AND #Events.%X12 AND NOT #ev THEN #Events.%X12 := FALSE; END_IF;
END_REGION

REGION Network 21: Сервисный режим
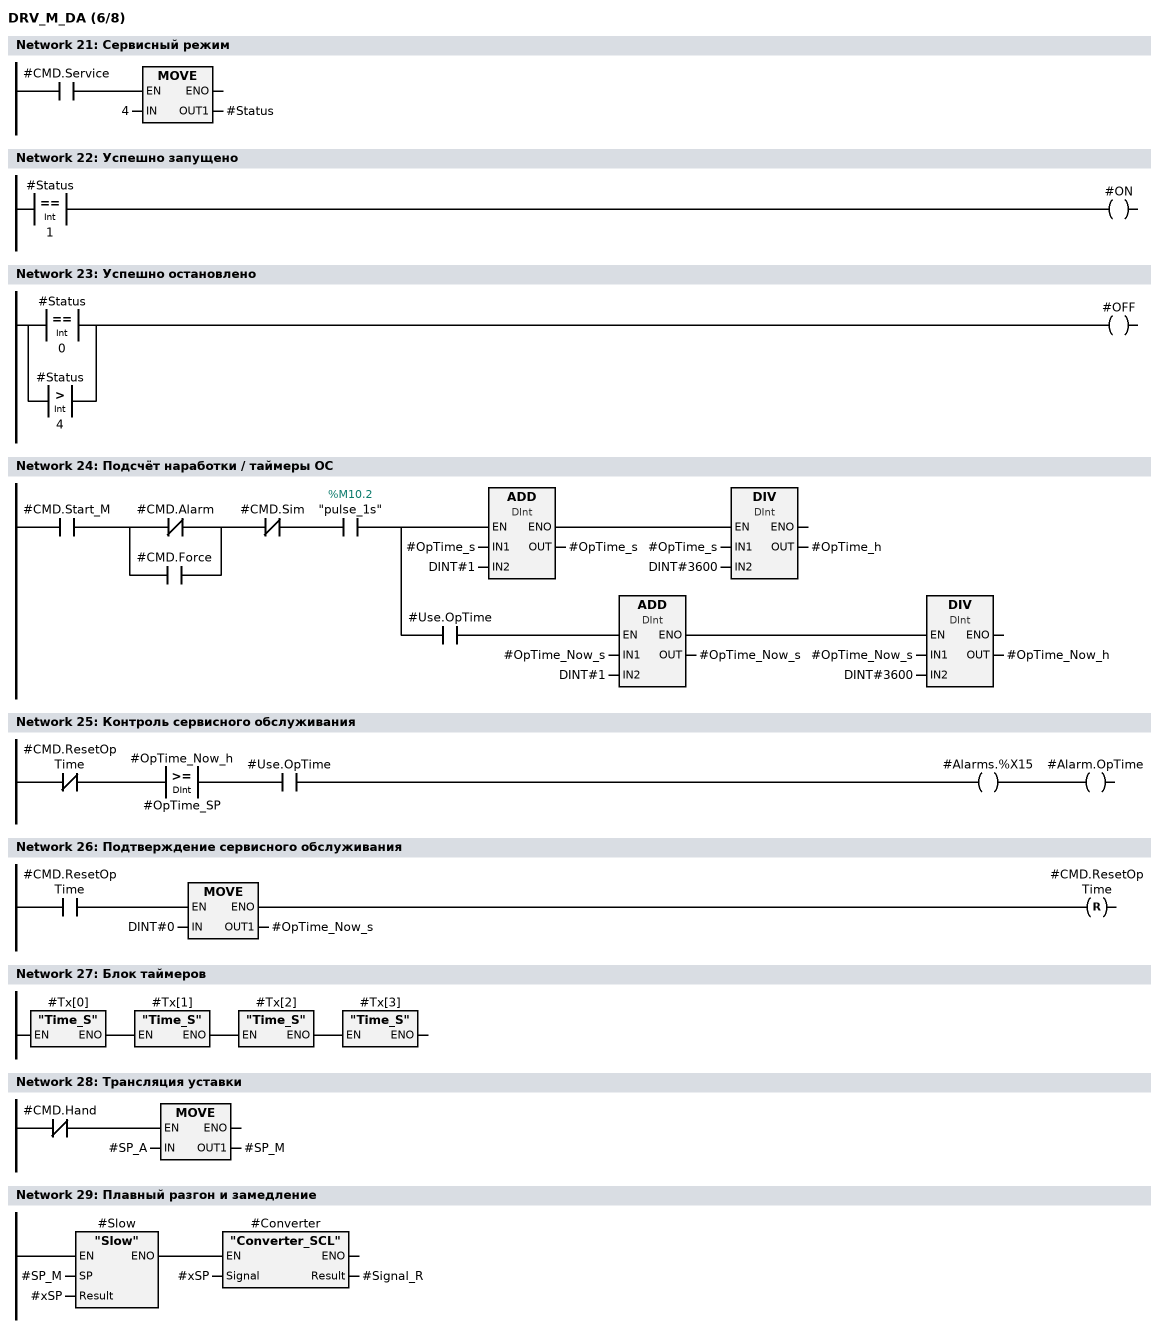
   RUNG wire#powerrail
      Contact( #CMD.Service )
      { S7_GenerateENO := "TRUE" } Move(in := 4, out1 => #Status)
   END_RUNG
   // the same network as SCL:
   IF #CMD.Service THEN #Status := 4; END_IF;
END_REGION

REGION Network 22: Успешно запущено
   RUNG wire#powerrail
      { S7_Templates := "SrcType := Int" } EQ_Contact(in1 := #Status, in2 := 1)
      Coil( #ON )
   END_RUNG
   // the same network as SCL:
   #ON := #Status = 1;
END_REGION

REGION Network 23: Успешно остановлено
   RUNG wire#powerrail
      { S7_Templates := "SrcType := Int" } EQ_Contact(in1 := #Status, in2 := 0)
      wire#w1
      Coil( #OFF )
   END_RUNG
   RUNG wire#powerrail
      { S7_Templates := "SrcType := Int" } GT_Contact(in1 := #Status, in2 := 4)
   END_RUNG wire#w1
   // the same network as SCL:
   #OFF := (#Status = 0) OR (#Status > 4);
END_REGION

REGION Network 24: Подсчёт наработки / таймеры ОС
   RUNG wire#powerrail
      Contact( #CMD.Start_M )
      wire#w1
      I_Contact( #CMD.Alarm )
      wire#w2
      I_Contact( #CMD.Sim )
      Contact( "pulse_1s" )
      wire#w3
      { S7_Templates := "SrcType := DInt"; S7_GenerateENO := "TRUE" } Add(in1 := #OpTime_s, in2 := DINT#1, out => #OpTime_s)
      { S7_Templates := "SrcType := DInt"; S7_GenerateENO := "TRUE" } Div(in1 := #OpTime_s, in2 := DINT#3600, out => #OpTime_h)
   END_RUNG
   RUNG wire#w1
      Contact( #CMD.Force )
   END_RUNG wire#w2
   RUNG wire#w3
      Contact( #Use.OpTime )
      { S7_Templates := "SrcType := DInt"; S7_GenerateENO := "TRUE" } Add(in1 := #OpTime_Now_s, in2 := DINT#1, out => #OpTime_Now_s)
      { S7_Templates := "SrcType := DInt"; S7_GenerateENO := "TRUE" } Div(in1 := #OpTime_Now_s, in2 := DINT#3600, out => #OpTime_Now_h)
   END_RUNG
   // the same network as SCL:
   // ENO of a box is taken as its EN; it also drops when the box reports an error
   #_w1 := #CMD.Start_M AND (NOT #CMD.Alarm OR #CMD.Force) AND NOT #CMD.Sim AND "pulse_1s";
   IF #_w1 THEN
       #OpTime_s := #OpTime_s + DINT#1;
       #OpTime_h := #OpTime_s / DINT#3600;
   END_IF;
   IF #_w1 AND #Use.OpTime THEN
       #OpTime_Now_s := #OpTime_Now_s + DINT#1;
       #OpTime_Now_h := #OpTime_Now_s / DINT#3600;
   END_IF;
END_REGION

REGION Network 25: Контроль сервисного обслуживания
   RUNG wire#powerrail
      I_Contact( #CMD.ResetOpTime )
      { S7_Templates := "SrcType := DInt" } GE_Contact(in1 := #OpTime_Now_h, in2 := #OpTime_SP)
      Contact( #Use.OpTime )
      Coil( #Alarms.%X15 )
      Coil( #Alarm.OpTime )
   END_RUNG
   // the same network as SCL:
   #Alarms.%X15 := NOT #CMD.ResetOpTime AND (#OpTime_Now_h >= #OpTime_SP) AND #Use.OpTime;
   #Alarm.OpTime := #Alarms.%X15;
END_REGION

REGION Network 26: Подтверждение сервисного обслуживания
   RUNG wire#powerrail
      Contact( #CMD.ResetOpTime )
      { S7_GenerateENO := "TRUE" } Move(in := DINT#0, out1 => #OpTime_Now_s)
      R_Coil( #CMD.ResetOpTime )
   END_RUNG
   // the same network as SCL:
   // ENO of a box is taken as its EN; it also drops when the box reports an error
   IF #CMD.ResetOpTime THEN
       #OpTime_Now_s := DINT#0;
       #CMD.ResetOpTime := FALSE;
   END_IF;
END_REGION

REGION Network 27: Блок таймеров
   RUNG wire#powerrail
      #Tx[0]()
      #Tx[1]()
      #Tx[2]()
      #Tx[3]()
   END_RUNG
   // the same network as SCL:
   #Tx[0](ENO => #_w1);   // "Time_S"
   #Tx[1](EN := #_w1, ENO => #_w2);   // "Time_S"
   #Tx[2](EN := #_w2, ENO => #_w3);   // "Time_S"
   IF #_w3 THEN
       #Tx[3]();   // "Time_S"
   END_IF;
END_REGION

REGION Network 28: Трансляция уставки
   RUNG wire#powerrail
      I_Contact( #CMD.Hand )
      Move(in := #SP_A, out1 => #SP_M)
   END_RUNG
   // the same network as SCL:
   IF NOT #CMD.Hand THEN #SP_M := #SP_A; END_IF;
END_REGION

REGION Network 29: Плавный разгон и замедление
   RUNG wire#powerrail
      #Slow(SP := #SP_M, Result := #xSP)
      #Converter(Signal := #xSP, Result => #Signal_R)
   END_RUNG
   // the same network as SCL:
   #Slow(SP := #SP_M, Result := #xSP, ENO => #_w1);   // "Slow"
   IF #_w1 THEN
       #Converter(Signal := #xSP, Result => #Signal_R);   // "Converter_SCL"
   END_IF;
END_REGION

REGION Network 30: Выходной аналоговый сигнал
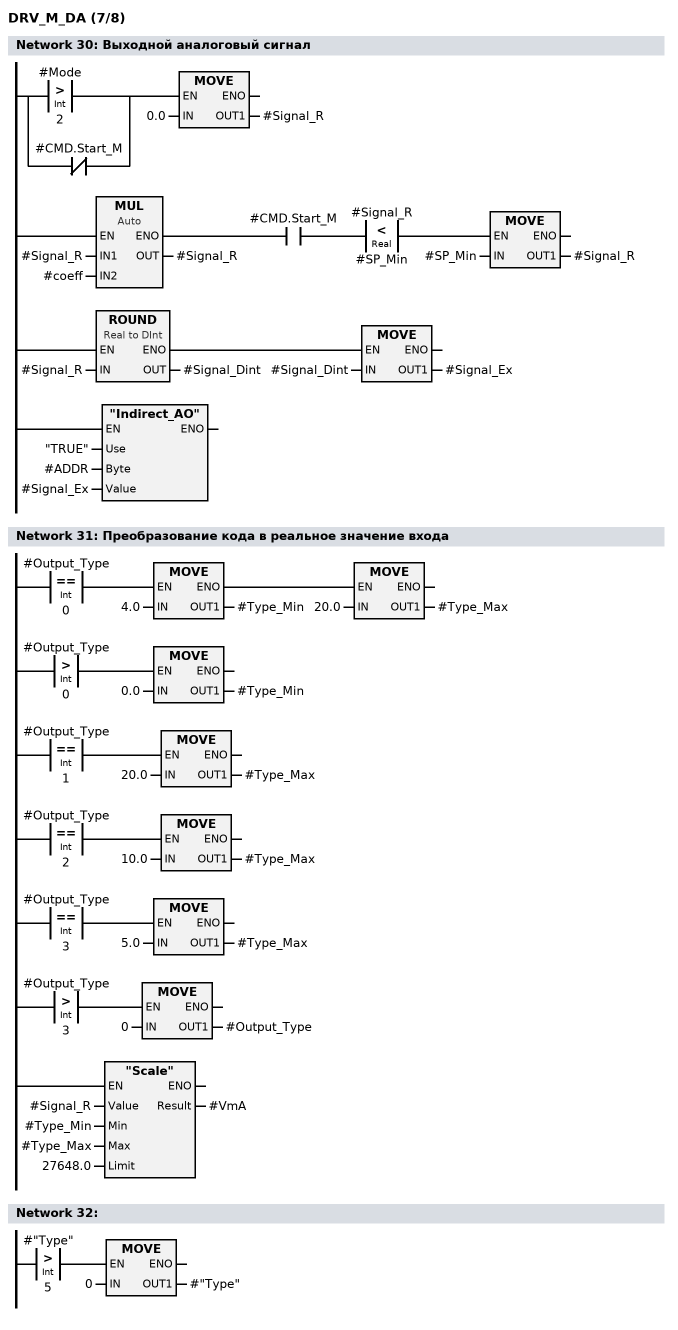
   RUNG wire#powerrail
      { S7_Templates := "SrcType := Int" } GT_Contact(in1 := #Mode, in2 := 2)
      wire#w1
      Move(in := 0.0, out1 => #Signal_R)
   END_RUNG
   RUNG wire#powerrail
      I_Contact( #CMD.Start_M )
   END_RUNG wire#w1
   RUNG wire#powerrail
      Mul(in1 := #Signal_R, in2 := #coeff, out => #Signal_R)
      Contact( #CMD.Start_M )
      { S7_Templates := "SrcType := Real" } LT_Contact(in1 := #Signal_R, in2 := #SP_Min)
      Move(in := #SP_Min, out1 => #Signal_R)
   END_RUNG
   RUNG wire#powerrail
      { S7_Templates := "[SrcType := Real, DestType := DInt]"; S7_GenerateENO := "TRUE" } Round(in := #Signal_R, out => #Signal_Dint)
      Move(in := #Signal_Dint, out1 => #Signal_Ex)
   END_RUNG
   RUNG wire#powerrail
      "Indirect_AO"(Use := "TRUE", "Byte" := #ADDR, Value := #Signal_Ex)
   END_RUNG
   // the same network as SCL:
   // ENO of a box is taken as its EN; it also drops when the box reports an error
   IF (#Mode > 2) OR NOT #CMD.Start_M THEN #Signal_R := 0.0; END_IF;
   #Signal_R := #Signal_R * #coeff;
   IF #CMD.Start_M AND (#Signal_R < #SP_Min) THEN #Signal_R := #SP_Min; END_IF;
   #Signal_Dint := ROUND(#Signal_R);
   #Signal_Ex := #Signal_Dint;
   "Indirect_AO"(Use := "TRUE", "Byte" := #ADDR, Value := #Signal_Ex);
END_REGION

REGION Network 31: Преобразование кода в реальное значение входа
   RUNG wire#powerrail
      { S7_Templates := "SrcType := Int" } EQ_Contact(in1 := #Output_Type, in2 := 0)
      Move(in := 4.0, out1 => #Type_Min)
      Move(in := 20.0, out1 => #Type_Max)
   END_RUNG
   RUNG wire#powerrail
      { S7_Templates := "SrcType := Int" } GT_Contact(in1 := #Output_Type, in2 := 0)
      Move(in := 0.0, out1 => #Type_Min)
   END_RUNG
   RUNG wire#powerrail
      { S7_Templates := "SrcType := Int" } EQ_Contact(in1 := #Output_Type, in2 := 1)
      Move(in := 20.0, out1 => #Type_Max)
   END_RUNG
   RUNG wire#powerrail
      { S7_Templates := "SrcType := Int" } EQ_Contact(in1 := #Output_Type, in2 := 2)
      Move(in := 10.0, out1 => #Type_Max)
   END_RUNG
   RUNG wire#powerrail
      { S7_Templates := "SrcType := Int" } EQ_Contact(in1 := #Output_Type, in2 := 3)
      Move(in := 5.0, out1 => #Type_Max)
   END_RUNG
   RUNG wire#powerrail
      { S7_Templates := "SrcType := Int" } GT_Contact(in1 := #Output_Type, in2 := 3)
      Move(in := 0, out1 => #Output_Type)
   END_RUNG
   RUNG wire#powerrail
      "Scale"(Value := #Signal_R, Min := #Type_Min, Max := #Type_Max, Limit := 27648.0, Result => #VmA)
   END_RUNG
   // the same network as SCL:
   IF #Output_Type = 0 THEN
       #Type_Min := 4.0;
       #Type_Max := 20.0;
   END_IF;
   IF #Output_Type > 0 THEN #Type_Min := 0.0; END_IF;
   IF #Output_Type = 1 THEN #Type_Max := 20.0; END_IF;
   IF #Output_Type = 2 THEN #Type_Max := 10.0; END_IF;
   IF #Output_Type = 3 THEN #Type_Max := 5.0; END_IF;
   IF #Output_Type > 3 THEN #Output_Type := 0; END_IF;
   "Scale"(Value := #Signal_R, Min := #Type_Min, Max := #Type_Max, Limit := 27648.0, Result => #VmA);
END_REGION

REGION Network 32
   RUNG wire#powerrail
      { S7_Templates := "SrcType := Int" } GT_Contact(in1 := #"Type", in2 := 5)
      Move(in := 0, out1 => #"Type")
   END_RUNG
   // the same network as SCL:
   IF #"Type" > 5 THEN #"Type" := 0; END_IF;
END_REGION

REGION Network 33: Метка времени
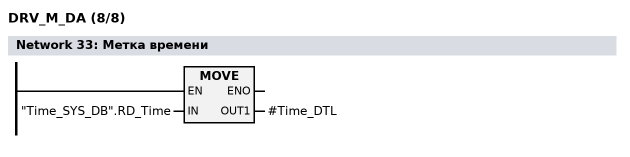
   RUNG wire#powerrail
      Move(in := "Time_SYS_DB".RD_Time, out1 => #Time_DTL)
   END_RUNG
   // the same network as SCL:
   #Time_DTL := "Time_SYS_DB".RD_Time;
END_REGION
END_FUNCTION_BLOCK

FUNCTION "drv_INV" : Void   // FC111, LAD
{ S7_Optimized_Access := 'FALSE' }
VERSION : 0.1
// stored: AutoNumber false, IsIECCheckEnabled false, SetENOAutomatically false, UDAEnableTagReadback false
   VAR_INPUT
      S : Bool;   // Сигнал
      I : Bool;   // Инверсия
   END_VAR
   VAR_IN_OUT
      R : Bool;   // Результат
   END_VAR
BEGIN

REGION Network 1: Инверсия сигнала
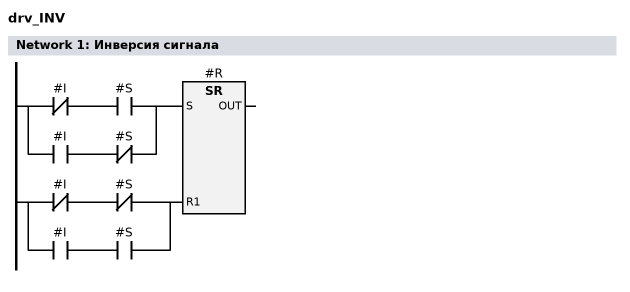
   RUNG wire#powerrail
      I_Contact( #I )
      Contact( #S )
      wire#w1
      S_SR(operand := #R, r1 := wire#w2)
   END_RUNG
   RUNG wire#powerrail
      Contact( #I )
      I_Contact( #S )
   END_RUNG wire#w1
   RUNG wire#powerrail
      I_Contact( #I )
      I_Contact( #S )
   END_RUNG wire#w2
   RUNG wire#powerrail
      Contact( #I )
      Contact( #S )
   END_RUNG wire#w2
   // the same network as SCL:
   IF (NOT #I AND #S) OR (#I AND NOT #S) THEN
       #R := TRUE;   // SR flip-flop
   END_IF;
   IF (NOT #I AND NOT #S) OR (#I AND #S) THEN #R := FALSE; END_IF;
END_REGION
END_FUNCTION

FUNCTION_BLOCK "Slow"   // FB151, LAD
{ S7_Optimized_Access := 'FALSE' }
VERSION : 0.1
// stored: AutoNumber false, IsIECCheckEnabled false, SetENOAutomatically false, UDAEnableTagReadback false
   VAR_INPUT
      SP : Real;   // Уставка
   END_VAR
   VAR_IN_OUT
      Result : Real;   // Управляющий сигнал
   END_VAR
   VAR DB_SPECIFIC
      Use_Up { S7_SetPoint := 'True'} : Bool;   // Использовать плавный разгон
      Use_Down { S7_SetPoint := 'True'} : Bool;   // Использовать плавное замедление
      Active : Bool;   // Идёт изменение уставки
      Active_Up : Bool;
      Active_Down : Bool;
      Step_Up { S7_SetPoint := 'True'} : Real := 0.125;   // Шаг плавного разгона
      Step_Down { S7_SetPoint := 'True'} : Real := 0.125;   // Шаг плавного замедления
   END_VAR
   VAR
      T_Up { S7_SetPoint := 'True'} : "Time_R";   // Таймер плавного разгона
      T_Down { S7_SetPoint := 'True'} : "Time_R";   // Таймер плавного замедления
   END_VAR
   VAR_TEMP
      Delta_Up : Real;   // Отклонение сигнала от уставки
      Delta_Down : Real;
   END_VAR
   VAR_TEMP   // added for the SCL form of the ladder/FBD networks
      _w1 : Bool;
      _w2 : Bool;
   END_VAR
BEGIN

REGION Network 1: Не используется
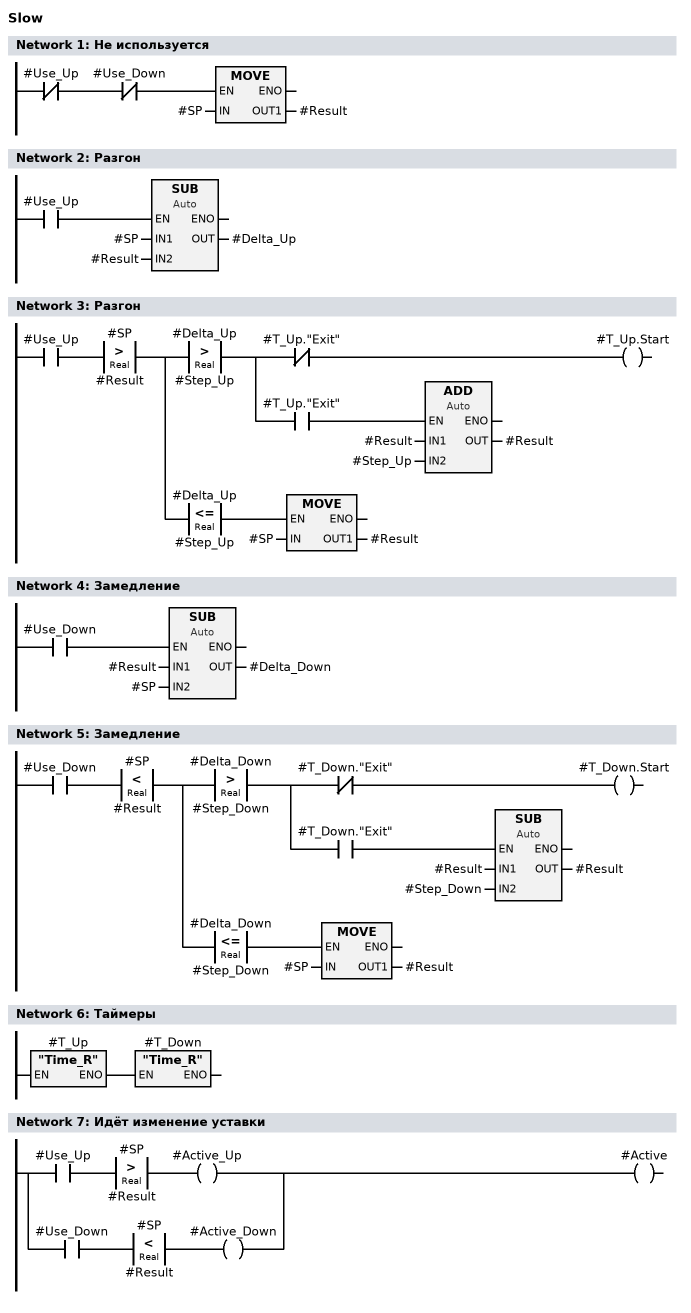
   RUNG wire#powerrail
      I_Contact( #Use_Up )
      I_Contact( #Use_Down )
      Move(in := #SP, out1 => #Result)
   END_RUNG
   // the same network as SCL:
   IF NOT #Use_Up AND NOT #Use_Down THEN #Result := #SP; END_IF;
END_REGION

REGION Network 2: Разгон
   RUNG wire#powerrail
      Contact( #Use_Up )
      Sub(in1 := #SP, in2 := #Result, out => #Delta_Up)
   END_RUNG
   // the same network as SCL:
   IF #Use_Up THEN #Delta_Up := #SP - #Result; END_IF;
END_REGION

REGION Network 3: Разгон
   RUNG wire#powerrail
      Contact( #Use_Up )
      { S7_Templates := "SrcType := Real" } GT_Contact(in1 := #SP, in2 := #Result)
      wire#w1
      { S7_Templates := "SrcType := Real" } GT_Contact(in1 := #Delta_Up, in2 := #Step_Up)
      wire#w2
      I_Contact( #T_Up."Exit" )
      Coil( #T_Up.Start )
   END_RUNG
   RUNG wire#w2
      Contact( #T_Up."Exit" )
      Add(in1 := #Result, in2 := #Step_Up, out => #Result)
   END_RUNG
   RUNG wire#w1
      { S7_Templates := "SrcType := Real" } LE_Contact(in1 := #Delta_Up, in2 := #Step_Up)
      Move(in := #SP, out1 => #Result)
   END_RUNG
   // the same network as SCL:
   #_w1 := #Use_Up AND (#SP > #Result);
   #_w2 := #_w1 AND (#Delta_Up > #Step_Up);
   #T_Up.Start := #_w2 AND NOT #T_Up."Exit";
   IF #_w2 AND #T_Up."Exit" THEN #Result := #Result + #Step_Up; END_IF;
   IF #_w1 AND (#Delta_Up <= #Step_Up) THEN #Result := #SP; END_IF;
END_REGION

REGION Network 4: Замедление
   RUNG wire#powerrail
      Contact( #Use_Down )
      Sub(in1 := #Result, in2 := #SP, out => #Delta_Down)
   END_RUNG
   // the same network as SCL:
   IF #Use_Down THEN #Delta_Down := #Result - #SP; END_IF;
END_REGION

REGION Network 5: Замедление
   RUNG wire#powerrail
      Contact( #Use_Down )
      { S7_Templates := "SrcType := Real" } LT_Contact(in1 := #SP, in2 := #Result)
      wire#w1
      { S7_Templates := "SrcType := Real" } GT_Contact(in1 := #Delta_Down, in2 := #Step_Down)
      wire#w2
      I_Contact( #T_Down."Exit" )
      Coil( #T_Down.Start )
   END_RUNG
   RUNG wire#w2
      Contact( #T_Down."Exit" )
      Sub(in1 := #Result, in2 := #Step_Down, out => #Result)
   END_RUNG
   RUNG wire#w1
      { S7_Templates := "SrcType := Real" } LE_Contact(in1 := #Delta_Down, in2 := #Step_Down)
      Move(in := #SP, out1 => #Result)
   END_RUNG
   // the same network as SCL:
   #_w1 := #Use_Down AND (#SP < #Result);
   #_w2 := #_w1 AND (#Delta_Down > #Step_Down);
   #T_Down.Start := #_w2 AND NOT #T_Down."Exit";
   IF #_w2 AND #T_Down."Exit" THEN #Result := #Result - #Step_Down; END_IF;
   IF #_w1 AND (#Delta_Down <= #Step_Down) THEN #Result := #SP; END_IF;
END_REGION

REGION Network 6: Таймеры
   RUNG wire#powerrail
      #T_Up()
      #T_Down()
   END_RUNG
   // the same network as SCL:
   #T_Up(ENO => #_w1);   // "Time_R"
   IF #_w1 THEN
       #T_Down();   // "Time_R"
   END_IF;
END_REGION

REGION Network 7: Идёт изменение уставки
   RUNG wire#powerrail
      Contact( #Use_Up )
      { S7_Templates := "SrcType := Real" } GT_Contact(in1 := #SP, in2 := #Result)
      Coil( #Active_Up )
      wire#w1
      Coil( #Active )
   END_RUNG
   RUNG wire#powerrail
      Contact( #Use_Down )
      { S7_Templates := "SrcType := Real" } LT_Contact(in1 := #SP, in2 := #Result)
      Coil( #Active_Down )
   END_RUNG wire#w1
   // the same network as SCL:
   #Active_Up := #Use_Up AND (#SP > #Result);
   #Active_Down := #Use_Down AND (#SP < #Result);
   #Active := #Active_Up OR #Active_Down;
END_REGION
END_FUNCTION_BLOCK

FUNCTION_BLOCK "Converter_SCL"
{ S7_Optimized_Access := 'FALSE' }
VERSION : 0.1
   VAR_INPUT 
      Signal : Real;
   END_VAR

   VAR_OUTPUT 
      Result : Real;
   END_VAR

   VAR 
      Lim_High { S7_SetPoint := 'True'} : Bool;
      Lim_Low { S7_SetPoint := 'True'} : Bool;
      Inverse { S7_SetPoint := 'True'} : Bool;
      Min_In { S7_SetPoint := 'True'} : Real;   // Минимальный входной сигнал
      Min_Out { S7_SetPoint := 'True'} : Real;   // Минимальный выходной сигнал
      Max_In { S7_SetPoint := 'True'} : Real;   // Максимальный входной сигнал
      Max_Out { S7_SetPoint := 'True'} : Real;   // Максимальный выходной сигнал
   END_VAR

   VAR_TEMP 
      Buffer : Real;
      Range_In : Real;
      Range_Out : Real;
      RR_Scale : Real;
      Value_Min : Real;
      Value_Max : Real;
   END_VAR


BEGIN
	//Диапазон входного сигнала
	IF #Min_In >= 0 THEN
	    #Range_In := #Max_In - #Min_In;
	ELSE
	    #Range_In := #Max_In + ABS(#Min_In);
	END_IF;
	
	//Диапазон выходного сигнала
	#Inverse := FALSE;
	IF #Min_Out >= 0 AND #Max_Out >= 0 THEN
	    IF #Max_Out > #Min_Out THEN
	        #Range_Out := #Max_Out - #Min_Out;
	        #Value_Min := #Min_Out;
	        #Value_Max := #Max_Out;
	    END_IF;
	    IF #Max_Out < #Min_Out THEN
	        #Range_Out := #Min_Out - #Max_Out;
	        #Value_Min := #Max_Out;
	        #Value_Max := #Min_Out;
	        #Inverse := TRUE;
	    END_IF;
	END_IF;
	IF #Min_Out < 0 AND #Max_Out >= 0 THEN
	    #Range_Out := #Max_Out + ABS(#Min_Out);
	END_IF;
	IF #Min_Out < 0 AND #Max_Out < 0 THEN
	    #Range_Out := ABS(#Max_Out) + ABS(#Min_Out);
	END_IF;
	
	//Соотношение диапазонов
	IF #Range_Out <> 0 THEN
	    #RR_Scale := #Range_In / #Range_Out;
	END_IF;
	
	//Линеаризация
	IF #RR_Scale <> 0 THEN
	    #Buffer := (#Signal - #Min_In) / #RR_Scale;
	END_IF;
	//Коррекция
	#Buffer := #Buffer + #Value_Min;
	
	//Инверсия
	IF #Inverse THEN
	    #Buffer := #Value_Max - #Buffer;
	END_IF;
	
	//Ограничение снизу
	IF #Buffer < #Value_Min THEN
	    #Buffer := #Value_Min;
	END_IF;
	
	//Ограничение сверху
	IF #Buffer > #Value_Max THEN
	    #Buffer := #Value_Max;
	END_IF;
	
	//Вывод значения
	#Result := #Buffer;
END_FUNCTION_BLOCK

FUNCTION "FC_DRV_End" : Void   // FC101, LAD
{ S7_Optimized_Access := 'FALSE' }
VERSION : 0.1
// stored: AutoNumber false, IsIECCheckEnabled false, SetENOAutomatically false, UDAEnableTagReadback false
   VAR_TEMP
      ev : Bool;
   END_VAR
   VAR_TEMP   // added for the SCL form of the ladder/FBD networks
      _w1 : Bool;
      _w2 : Bool;
      _w3 : Bool;
      _w4 : Bool;
      _w5 : Bool;
      _w6 : Bool;
      _w7 : Bool;
      _w8 : Bool;
   END_VAR
BEGIN

REGION Network 1: Одно из устройств нижнего уровня в ручном режиме
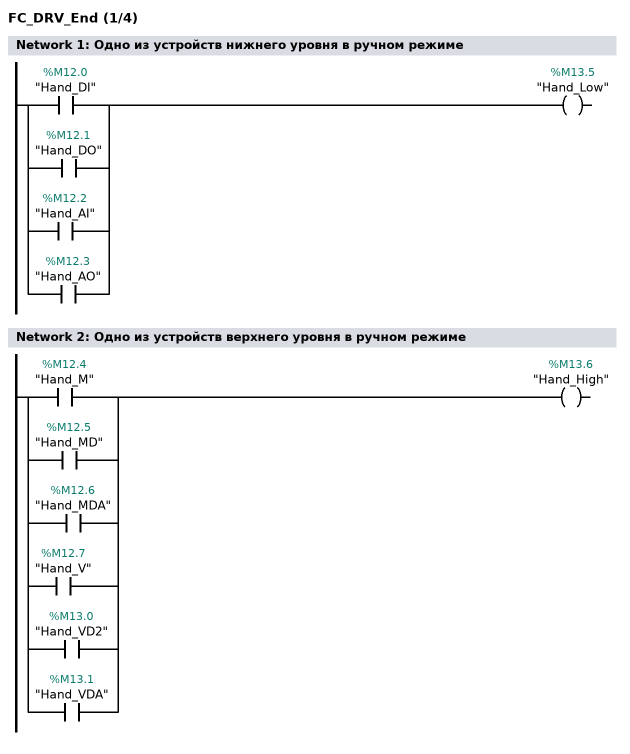
   RUNG wire#powerrail
      Contact( "Hand_DI" )
      wire#w1
      Coil( "Hand_Low" )
   END_RUNG
   RUNG wire#powerrail
      Contact( "Hand_DO" )
   END_RUNG wire#w1
   RUNG wire#powerrail
      Contact( "Hand_AI" )
   END_RUNG wire#w1
   RUNG wire#powerrail
      Contact( "Hand_AO" )
   END_RUNG wire#w1
   // the same network as SCL:
   "Hand_Low" := "Hand_DI" OR "Hand_DO" OR "Hand_AI" OR "Hand_AO";
END_REGION

REGION Network 2: Одно из устройств верхнего уровня в ручном режиме
   RUNG wire#powerrail
      Contact( "Hand_M" )
      wire#w1
      Coil( "Hand_High" )
   END_RUNG
   RUNG wire#powerrail
      Contact( "Hand_MD" )
   END_RUNG wire#w1
   RUNG wire#powerrail
      Contact( "Hand_MDA" )
   END_RUNG wire#w1
   RUNG wire#powerrail
      Contact( "Hand_V" )
   END_RUNG wire#w1
   RUNG wire#powerrail
      Contact( "Hand_VD2" )
   END_RUNG wire#w1
   RUNG wire#powerrail
      Contact( "Hand_VDA" )
   END_RUNG wire#w1
   // the same network as SCL:
   "Hand_High" := "Hand_M" OR "Hand_MD" OR "Hand_MDA" OR "Hand_V" OR "Hand_VD2" OR "Hand_VDA";
END_REGION

REGION Network 3: Сбор и сброс статусов ручного режима
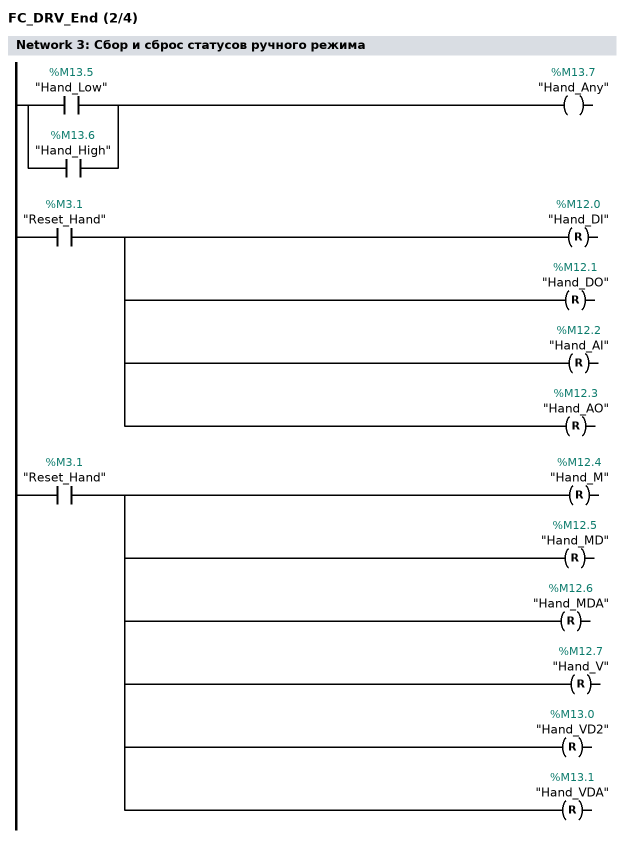
   RUNG wire#powerrail
      Contact( "Hand_Low" )
      wire#w1
      Coil( "Hand_Any" )
   END_RUNG
   RUNG wire#powerrail
      Contact( "Hand_High" )
   END_RUNG wire#w1
   RUNG wire#powerrail
      Contact( "Reset_Hand" )
      wire#w2
      R_Coil( "Hand_DI" )
   END_RUNG
   RUNG wire#w2
      R_Coil( "Hand_DO" )
   END_RUNG
   RUNG wire#w2
      R_Coil( "Hand_AI" )
   END_RUNG
   RUNG wire#w2
      R_Coil( "Hand_AO" )
   END_RUNG
   RUNG wire#powerrail
      Contact( "Reset_Hand" )
      wire#w3
      R_Coil( "Hand_M" )
   END_RUNG
   RUNG wire#w3
      R_Coil( "Hand_MD" )
   END_RUNG
   RUNG wire#w3
      R_Coil( "Hand_MDA" )
   END_RUNG
   RUNG wire#w3
      R_Coil( "Hand_V" )
   END_RUNG
   RUNG wire#w3
      R_Coil( "Hand_VD2" )
   END_RUNG
   RUNG wire#w3
      R_Coil( "Hand_VDA" )
   END_RUNG
   // the same network as SCL:
   "Hand_Any" := "Hand_Low" OR "Hand_High";
   IF "Reset_Hand" THEN
       "Hand_DI" := FALSE;
       "Hand_DO" := FALSE;
       "Hand_AI" := FALSE;
       "Hand_AO" := FALSE;
       "Hand_M" := FALSE;
       "Hand_MD" := FALSE;
       "Hand_MDA" := FALSE;
       "Hand_V" := FALSE;
       "Hand_VD2" := FALSE;
       "Hand_VDA" := FALSE;
   END_IF;
END_REGION

REGION Network 4
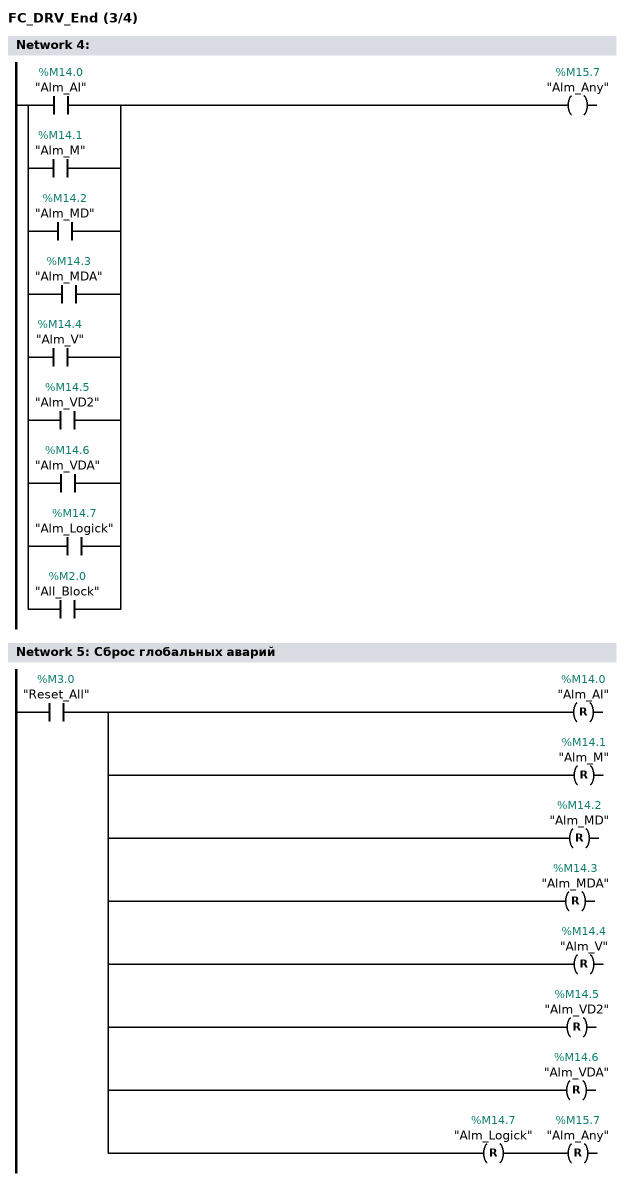
   RUNG wire#powerrail
      Contact( "Alm_AI" )
      wire#w1
      Coil( "Alm_Any" )
   END_RUNG
   RUNG wire#powerrail
      Contact( "Alm_M" )
   END_RUNG wire#w1
   RUNG wire#powerrail
      Contact( "Alm_MD" )
   END_RUNG wire#w1
   RUNG wire#powerrail
      Contact( "Alm_MDA" )
   END_RUNG wire#w1
   RUNG wire#powerrail
      Contact( "Alm_V" )
   END_RUNG wire#w1
   RUNG wire#powerrail
      Contact( "Alm_VD2" )
   END_RUNG wire#w1
   RUNG wire#powerrail
      Contact( "Alm_VDA" )
   END_RUNG wire#w1
   RUNG wire#powerrail
      Contact( "Alm_Logick" )
   END_RUNG wire#w1
   RUNG wire#powerrail
      Contact( "All_Block" )
   END_RUNG wire#w1
   // the same network as SCL:
   "Alm_Any" := "Alm_AI" OR "Alm_M" OR "Alm_MD" OR "Alm_MDA" OR "Alm_V" OR "Alm_VD2" OR "Alm_VDA" OR "Alm_Logick" OR "All_Block";
END_REGION

REGION Network 5: Сброс глобальных аварий
   RUNG wire#powerrail
      Contact( "Reset_All" )
      wire#w1
      R_Coil( "Alm_AI" )
   END_RUNG
   RUNG wire#w1
      R_Coil( "Alm_M" )
   END_RUNG
   RUNG wire#w1
      R_Coil( "Alm_MD" )
   END_RUNG
   RUNG wire#w1
      R_Coil( "Alm_MDA" )
   END_RUNG
   RUNG wire#w1
      R_Coil( "Alm_V" )
   END_RUNG
   RUNG wire#w1
      R_Coil( "Alm_VD2" )
   END_RUNG
   RUNG wire#w1
      R_Coil( "Alm_VDA" )
   END_RUNG
   RUNG wire#w1
      R_Coil( "Alm_Logick" )
      R_Coil( "Alm_Any" )
   END_RUNG
   // the same network as SCL:
   IF "Reset_All" THEN
       "Alm_AI" := FALSE;
       "Alm_M" := FALSE;
       "Alm_MD" := FALSE;
       "Alm_MDA" := FALSE;
       "Alm_V" := FALSE;
       "Alm_VD2" := FALSE;
       "Alm_VDA" := FALSE;
       "Alm_Logick" := FALSE;
       "Alm_Any" := FALSE;
   END_IF;
END_REGION

REGION Network 6: Основные события
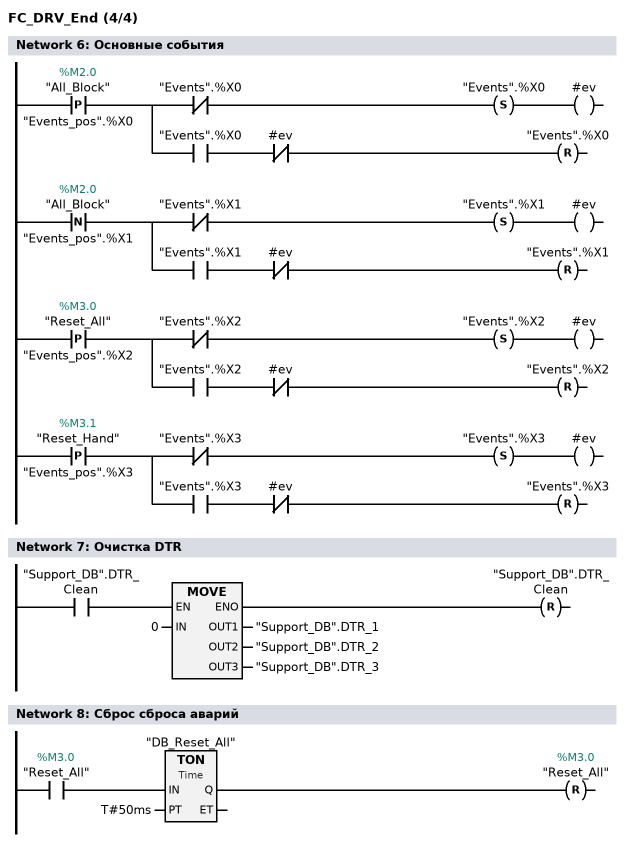
   RUNG wire#powerrail
      P_Contact(operand := "All_Block", bit := "Events_pos".%X0)
      wire#w1
      I_Contact( "Events".%X0 )
      S_Coil( "Events".%X0 )
      Coil( #ev )
   END_RUNG
   RUNG wire#w1
      Contact( "Events".%X0 )
      I_Contact( #ev )
      R_Coil( "Events".%X0 )
   END_RUNG
   RUNG wire#powerrail
      N_Contact(operand := "All_Block", bit := "Events_pos".%X1)
      wire#w2
      I_Contact( "Events".%X1 )
      S_Coil( "Events".%X1 )
      Coil( #ev )
   END_RUNG
   RUNG wire#w2
      Contact( "Events".%X1 )
      I_Contact( #ev )
      R_Coil( "Events".%X1 )
   END_RUNG
   RUNG wire#powerrail
      P_Contact(operand := "Reset_All", bit := "Events_pos".%X2)
      wire#w3
      I_Contact( "Events".%X2 )
      S_Coil( "Events".%X2 )
      Coil( #ev )
   END_RUNG
   RUNG wire#w3
      Contact( "Events".%X2 )
      I_Contact( #ev )
      R_Coil( "Events".%X2 )
   END_RUNG
   RUNG wire#powerrail
      P_Contact(operand := "Reset_Hand", bit := "Events_pos".%X3)
      wire#w4
      I_Contact( "Events".%X3 )
      S_Coil( "Events".%X3 )
      Coil( #ev )
   END_RUNG
   RUNG wire#w4
      Contact( "Events".%X3 )
      I_Contact( #ev )
      R_Coil( "Events".%X3 )
   END_RUNG
   // the same network as SCL:
   #_w1 := "All_Block" AND NOT "Events_pos".%X0;   // rising edge of "All_Block"
   "Events_pos".%X0 := "All_Block";
   #_w2 := #_w1 AND NOT "Events".%X0;
   IF #_w2 THEN "Events".%X0 := TRUE; END_IF;
   #ev := #_w2;
   IF #_w1 AND "Events".%X0 AND NOT #ev THEN "Events".%X0 := FALSE; END_IF;
   #_w3 := NOT "All_Block" AND "Events_pos".%X1;   // falling edge of "All_Block"
   "Events_pos".%X1 := "All_Block";
   #_w4 := #_w3 AND NOT "Events".%X1;
   IF #_w4 THEN "Events".%X1 := TRUE; END_IF;
   #ev := #_w4;
   IF #_w3 AND "Events".%X1 AND NOT #ev THEN "Events".%X1 := FALSE; END_IF;
   #_w5 := "Reset_All" AND NOT "Events_pos".%X2;   // rising edge of "Reset_All"
   "Events_pos".%X2 := "Reset_All";
   #_w6 := #_w5 AND NOT "Events".%X2;
   IF #_w6 THEN "Events".%X2 := TRUE; END_IF;
   #ev := #_w6;
   IF #_w5 AND "Events".%X2 AND NOT #ev THEN "Events".%X2 := FALSE; END_IF;
   #_w7 := "Reset_Hand" AND NOT "Events_pos".%X3;   // rising edge of "Reset_Hand"
   "Events_pos".%X3 := "Reset_Hand";
   #_w8 := #_w7 AND NOT "Events".%X3;
   IF #_w8 THEN "Events".%X3 := TRUE; END_IF;
   #ev := #_w8;
   IF #_w7 AND "Events".%X3 AND NOT #ev THEN "Events".%X3 := FALSE; END_IF;
END_REGION

REGION Network 7: Очистка DTR
   RUNG wire#powerrail
      Contact( "Support_DB".DTR_Clean )
      Move(in := 0, out1 => "Support_DB".DTR_1, out2 => "Support_DB".DTR_2, out3 => "Support_DB".DTR_3)
      R_Coil( "Support_DB".DTR_Clean )
   END_RUNG
   // the same network as SCL:
   IF "Support_DB".DTR_Clean THEN
       "Support_DB".DTR_1 := 0;
       "Support_DB".DTR_2 := 0;
       "Support_DB".DTR_3 := 0;
       "Support_DB".DTR_Clean := FALSE;
   END_IF;
END_REGION

REGION Network 8: Сброс сброса аварий
   RUNG wire#powerrail
      Contact( "Reset_All" )
      { S7_Templates := "time_type := Time" } "DB_Reset_All".TON(pt := T#50ms, et =>)
      R_Coil( "Reset_All" )
   END_RUNG
   // the same network as SCL:
   "DB_Reset_All".TON(IN := "Reset_All", PT := T#50ms);
   IF "DB_Reset_All".Q THEN "Reset_All" := FALSE; END_IF;
END_REGION
END_FUNCTION

ORGANIZATION_BLOCK "Cyclic interrupt"   // OB30, LAD, CyclicInterrupt
{ S7_Optimized_Access := 'TRUE' }
VERSION : 0.1
// stored: AutoNumber true, IsIECCheckEnabled false, SetENOAutomatically false
   VAR_INPUT
      Initial_Call : Bool;   // Initial call of this OB
      Event_Count : Int;   // Events discarded
   END_VAR
BEGIN

REGION Network 1
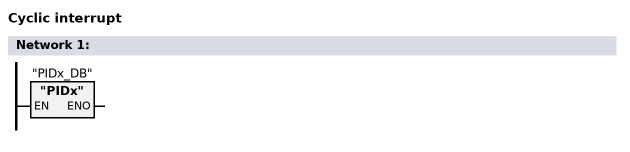
   RUNG wire#powerrail
      "PIDx_DB"()
   END_RUNG
   // the same network as SCL:
   "PIDx_DB"();   // "PIDx"
END_REGION
END_ORGANIZATION_BLOCK

FUNCTION_BLOCK "PIDx"   // FB260, LAD
{ S7_Optimized_Access := 'TRUE' }
VERSION : 0.1
// stored: AutoNumber false, IsIECCheckEnabled false, IsRetainMemResEnabled false, MemoryReserve 100, SetENOAutomatically false, UDAEnableTagReadback false
   VAR DB_SPECIFIC
      Time_DTL { S7_SetPoint := 'True'} : DTL;
   END_VAR
BEGIN

REGION Network 1
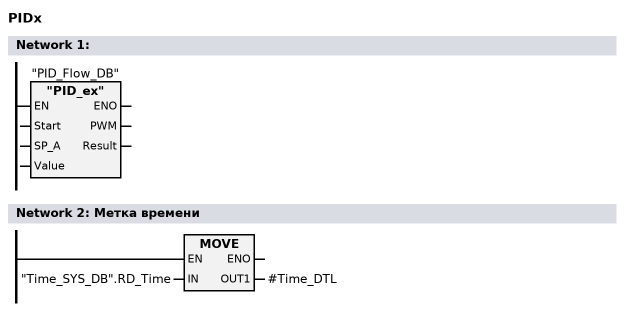
   RUNG wire#powerrail
      "PID_Flow_DB"(Start :=, SP_A :=, Value :=, PWM =>, Result =>)
   END_RUNG
   // the same network as SCL:
   "PID_Flow_DB"();   // "PID_ex"
END_REGION

REGION Network 2: Метка времени
   RUNG wire#powerrail
      Move(in := "Time_SYS_DB".RD_Time, out1 => #Time_DTL)
   END_RUNG
   // the same network as SCL:
   #Time_DTL := "Time_SYS_DB".RD_Time;
END_REGION
END_FUNCTION_BLOCK

FUNCTION_BLOCK "PID_ex"   // FB99, LAD
{ S7_Optimized_Access := 'FALSE' }
VERSION : 0.1
// stored: AutoNumber false, IsIECCheckEnabled false, SetENOAutomatically false, UDAEnableTagReadback false
   VAR_INPUT
      Start : Bool;
      SP_A : Real;   // Уставка
      Value : Real;   // Показания датчика
   END_VAR
   VAR_OUTPUT
      PWM : Bool;   // ШИМ-выход ПИД-регулятора
      Result : Real;   // Управляющее воздействие
   END_VAR
   VAR DB_SPECIFIC
      CMD { S7_SetPoint := 'True'} : "CMD";
      SP_M : Real;
      SP : Real;
      x { S7_SetPoint := 'True'} : Real := 1.0;   // Поправка уставки и датчика
      SP_x : Real;   // Домноженная уставка
      Value_x : Real;   // Домноженный датчик
      Buffer : Real;   // Промежуточное значение
      PID_Output : Real;   // Выход ПИД-регулятора
      PID_Hand : Real;   // Ручное задание выхода ПИД-регулятора
      Sys : Struct   // Системные параметры
         Err_Ack : Bool;   // Подтверждение аварии
         Alm_SP_H : Bool;   // Авария уставки - превышение
         Alm_SP_L : Bool;   // Авария уставки - занижение
         Alm_In_H : Bool;   // Авария датчика - превышение
         Alm_In_L : Bool;   // Авария датчика - занижение
         Activate : Bool;   // Активировать ПИД
         Error_code : DWord;   // Код аварии
         Warning_code : DWord;   // Код предупреждения
         "Type" : Int := 1;   // Режим работы
         State : Int;   // Состояние
         Mode : Int := 3;   // Режим
      END_STRUCT;
      Settings : Struct   // Рабочие параметры
         SP_P { S7_SetPoint := 'True'} : Real := 1.5;   // Коэффициент пропорциональности
         SP_Ti { S7_SetPoint := 'True'} : Real := 150.0;   // Время интегрирования
         SP_Td { S7_SetPoint := 'True'} : Real;   // Время дифференцирования
         SP_Cycle { S7_SetPoint := 'True'} : Real := 0.2;   // Время цикла
         Max_SP { S7_SetPoint := 'True'} : Real := 500.0;   // Максимальное значение уставки
         Min_SP { S7_SetPoint := 'True'} : Real := -500.0;   // Минимальное значение уставки
         Max_in { S7_SetPoint := 'True'} : Real := 500.0;   // Максимальное значение датчика
         Min_in { S7_SetPoint := 'True'} : Real := -500.0;   // Минимальное значение датчика
         Max_out { S7_SetPoint := 'True'} : Real := 100.0;   // Максимальное значение выхода
         Min_out { S7_SetPoint := 'True'} : Real := 0.0;   // Минимальное значение выхода
         DeadBand { S7_SetPoint := 'True'} : Real := 1.0;   // Мёртвая зона
         Max : Real;   // Верняя граница мёртвой зоны
         Min : Real;   // Нижняя граница мёртвой зоны
      END_STRUCT;
   END_VAR
   VAR
      PID { S7_SetPoint := 'True'} : PID_Compact;   // ПИД
      Converter : "Converter_SCL";   // Конвертер выхода
      Conveter_Back : "Converter_SCL";   // Конвертер Hand_SP в 0..100
      C { S7_SetPoint := 'True'} : "Time_R";   // Частота вызова ПИД на обработку
   END_VAR
   VAR DB_SPECIFIC
      pos : Array[0..15] of Bool;
   END_VAR
   VAR_TEMP
      x0 : Real;
   END_VAR
   // CMD.Start_A := true;
   // Converter.Max_In := 100.0;
   // Conveter_Back.Max_Out := 100.0;
   VAR_TEMP   // added for the SCL form of the ladder/FBD networks
      _w1 : Bool;
      _w2 : Bool;
   END_VAR
BEGIN

REGION Network 1: Сброс ПИД
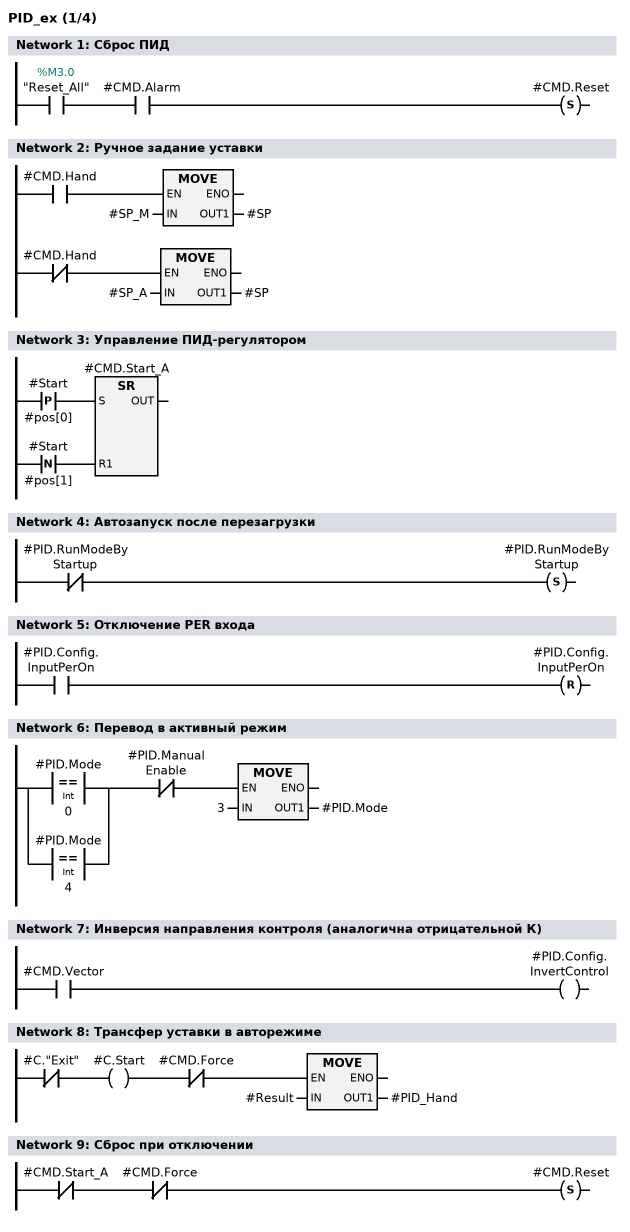
   RUNG wire#powerrail
      Contact( "Reset_All" )
      Contact( #CMD.Alarm )
      S_Coil( #CMD.Reset )
   END_RUNG
   // the same network as SCL:
   IF "Reset_All" AND #CMD.Alarm THEN #CMD.Reset := TRUE; END_IF;
END_REGION

REGION Network 2: Ручное задание уставки
   RUNG wire#powerrail
      Contact( #CMD.Hand )
      Move(in := #SP_M, out1 => #SP)
   END_RUNG
   RUNG wire#powerrail
      I_Contact( #CMD.Hand )
      Move(in := #SP_A, out1 => #SP)
   END_RUNG
   // the same network as SCL:
   IF #CMD.Hand THEN #SP := #SP_M; END_IF;
   IF NOT #CMD.Hand THEN #SP := #SP_A; END_IF;
END_REGION

REGION Network 3: Управление ПИД-регулятором
   RUNG wire#powerrail
      P_Contact(operand := #Start, bit := #pos[0])
      S_SR(operand := #CMD.Start_A, r1 := wire#w1)
   END_RUNG
   RUNG wire#powerrail
      N_Contact(operand := #Start, bit := #pos[1])
   END_RUNG wire#w1
   // the same network as SCL:
   #_w1 := #Start AND NOT #pos[0];   // rising edge of #Start
   #pos[0] := #Start;
   #_w2 := NOT #Start AND #pos[1];   // falling edge of #Start
   #pos[1] := #Start;
   IF #_w1 THEN
       #CMD.Start_A := TRUE;   // SR flip-flop
   END_IF;
   IF #_w2 THEN #CMD.Start_A := FALSE; END_IF;
END_REGION

REGION Network 4: Автозапуск после перезагрузки
   RUNG wire#powerrail
      I_Contact( #PID.RunModeByStartup )
      S_Coil( #PID.RunModeByStartup )
   END_RUNG
   // the same network as SCL:
   IF NOT #PID.RunModeByStartup THEN #PID.RunModeByStartup := TRUE; END_IF;
END_REGION

REGION Network 5: Отключение PER входа
   RUNG wire#powerrail
      Contact( #PID.Config.InputPerOn )
      R_Coil( #PID.Config.InputPerOn )
   END_RUNG
   // the same network as SCL:
   IF #PID.Config.InputPerOn THEN #PID.Config.InputPerOn := FALSE; END_IF;
END_REGION

REGION Network 6: Перевод в активный режим
   RUNG wire#powerrail
      { S7_Templates := "SrcType := Int" } EQ_Contact(in1 := #PID.Mode, in2 := 0)
      wire#w1
      I_Contact( #PID.ManualEnable )
      { S7_GenerateENO := "TRUE" } Move(in := 3, out1 => #PID.Mode)
   END_RUNG
   RUNG wire#powerrail
      { S7_Templates := "SrcType := Int" } EQ_Contact(in1 := #PID.Mode, in2 := 4)
   END_RUNG wire#w1
   // the same network as SCL:
   IF ((#PID.Mode = 0) OR (#PID.Mode = 4)) AND NOT #PID.ManualEnable THEN #PID.Mode := 3; END_IF;
END_REGION

REGION Network 7: Инверсия направления контроля (аналогична отрицательной К)
   RUNG wire#powerrail
      Contact( #CMD.Vector )
      Coil( #PID.Config.InvertControl )
   END_RUNG
   // the same network as SCL:
   #PID.Config.InvertControl := #CMD.Vector;
END_REGION

REGION Network 8: Трансфер уставки в авторежиме
   RUNG wire#powerrail
      I_Contact( #C."Exit" )
      Coil( #C.Start )
      I_Contact( #CMD.Force )
      Move(in := #Result, out1 => #PID_Hand)
   END_RUNG
   // the same network as SCL:
   #C.Start := NOT #C."Exit";
   IF NOT #C."Exit" AND NOT #CMD.Force THEN #PID_Hand := #Result; END_IF;
END_REGION

REGION Network 9: Сброс при отключении
   RUNG wire#powerrail
      I_Contact( #CMD.Start_A )
      I_Contact( #CMD.Force )
      S_Coil( #CMD.Reset )
   END_RUNG
   // the same network as SCL:
   IF NOT #CMD.Start_A AND NOT #CMD.Force THEN #CMD.Reset := TRUE; END_IF;
END_REGION

REGION Network 10: Активация после смены режима
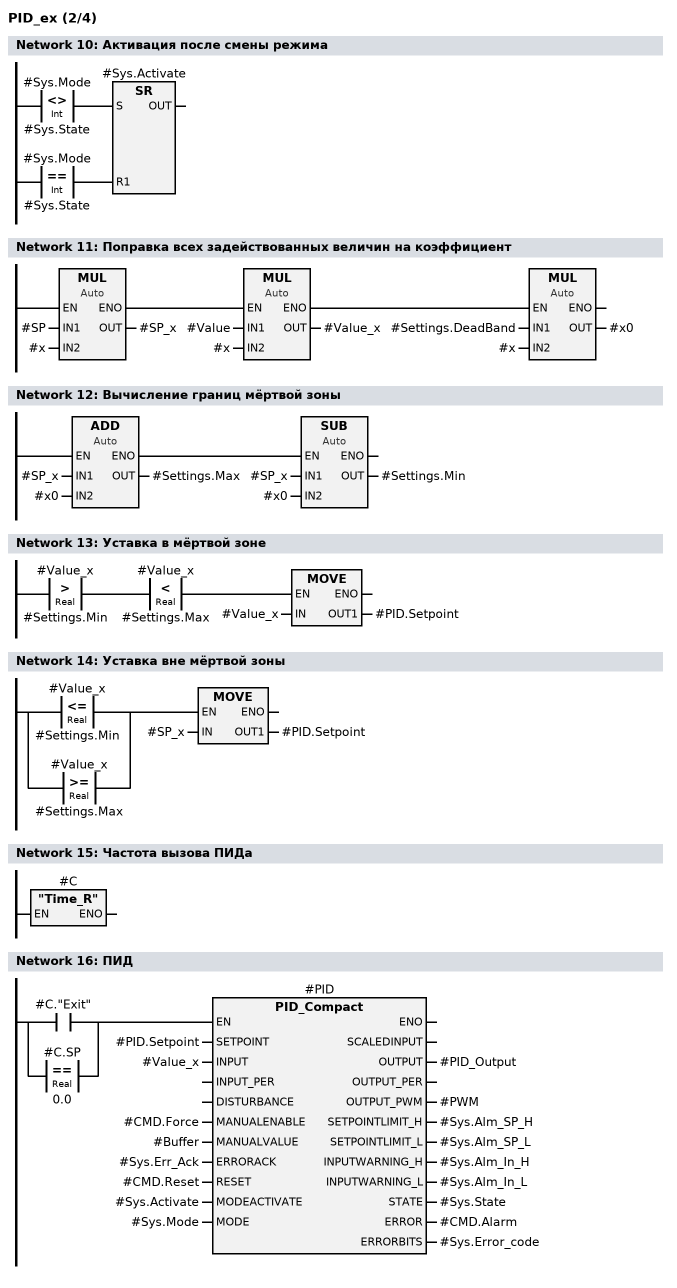
   RUNG wire#powerrail
      { S7_Templates := "SrcType := Int" } NE_Contact(in1 := #Sys.Mode, in2 := #Sys.State)
      S_SR(operand := #Sys.Activate, r1 := wire#w1)
   END_RUNG
   RUNG wire#powerrail
      { S7_Templates := "SrcType := Int" } EQ_Contact(in1 := #Sys.Mode, in2 := #Sys.State)
   END_RUNG wire#w1
   // the same network as SCL:
   IF #Sys.Mode <> #Sys.State THEN
       #Sys.Activate := TRUE;   // SR flip-flop
   END_IF;
   IF #Sys.Mode = #Sys.State THEN #Sys.Activate := FALSE; END_IF;
END_REGION

REGION Network 11: Поправка всех задействованных величин на коэффициент
   RUNG wire#powerrail
      Mul(in1 := #SP, in2 := #x, out => #SP_x)
      Mul(in1 := #Value, in2 := #x, out => #Value_x)
      Mul(in1 := #Settings.DeadBand, in2 := #x, out => #x0)
   END_RUNG
   // the same network as SCL:
   #SP_x := #SP * #x;
   #Value_x := #Value * #x;
   #x0 := #Settings.DeadBand * #x;
END_REGION

REGION Network 12: Вычисление границ мёртвой зоны
   RUNG wire#powerrail
      Add(in1 := #SP_x, in2 := #x0, out => #Settings.Max)
      Sub(in1 := #SP_x, in2 := #x0, out => #Settings.Min)
   END_RUNG
   // the same network as SCL:
   #Settings.Max := #SP_x + #x0;
   #Settings.Min := #SP_x - #x0;
END_REGION

REGION Network 13: Уставка в мёртвой зоне
   RUNG wire#powerrail
      { S7_Templates := "SrcType := Real" } GT_Contact(in1 := #Value_x, in2 := #Settings.Min)
      { S7_Templates := "SrcType := Real" } LT_Contact(in1 := #Value_x, in2 := #Settings.Max)
      Move(in := #Value_x, out1 => #PID.Setpoint)
   END_RUNG
   // the same network as SCL:
   IF (#Value_x > #Settings.Min) AND (#Value_x < #Settings.Max) THEN #PID.Setpoint := #Value_x; END_IF;
END_REGION

REGION Network 14: Уставка вне мёртвой зоны
   RUNG wire#powerrail
      { S7_Templates := "SrcType := Real" } LE_Contact(in1 := #Value_x, in2 := #Settings.Min)
      wire#w1
      Move(in := #SP_x, out1 => #PID.Setpoint)
   END_RUNG
   RUNG wire#powerrail
      { S7_Templates := "SrcType := Real" } GE_Contact(in1 := #Value_x, in2 := #Settings.Max)
   END_RUNG wire#w1
   // the same network as SCL:
   IF (#Value_x <= #Settings.Min) OR (#Value_x >= #Settings.Max) THEN #PID.Setpoint := #SP_x; END_IF;
END_REGION

REGION Network 15: Частота вызова ПИДа
   RUNG wire#powerrail
      #C()
   END_RUNG
   // the same network as SCL:
   #C();   // "Time_R"
END_REGION

REGION Network 16: ПИД
   RUNG wire#powerrail
      Contact( #C."Exit" )
      wire#w1
      #PID.PID_Compact(Setpoint := #PID.Setpoint, Input := #Value_x, Input_PER :=, Disturbance :=, ManualEnable := #CMD.Force, ManualValue := #Buffer, ErrorAck := #Sys.Err_Ack, Reset := #CMD.Reset, ModeActivate := #Sys.Activate, Mode := #Sys.Mode, ScaledInput =>, Output => #PID_Output, Output_PER =>, Output_PWM => #PWM, SetpointLimit_H => #Sys.Alm_SP_H, SetpointLimit_L => #Sys.Alm_SP_L, InputWarning_H => #Sys.Alm_In_H, InputWarning_L => #Sys.Alm_In_L, State => #Sys.State, Error => #CMD.Alarm, ErrorBits => #Sys.Error_code)
   END_RUNG
   RUNG wire#powerrail
      { S7_Templates := "SrcType := Real" } EQ_Contact(in1 := #C.SP, in2 := 0.0)
   END_RUNG wire#w1
   // the same network as SCL:
   IF #C."Exit" OR (#C.SP = 0.0) THEN
       #PID(Setpoint := #PID.Setpoint,   // PID_Compact
            Input := #Value_x,
            ManualEnable := #CMD.Force,
            ManualValue := #Buffer,
            ErrorAck := #Sys.Err_Ack,
            Reset := #CMD.Reset,
            ModeActivate := #Sys.Activate,
            Mode := #Sys.Mode,
            Output => #PID_Output,
            Output_PWM => #PWM,
            SetpointLimit_H => #Sys.Alm_SP_H,
            SetpointLimit_L => #Sys.Alm_SP_L,
            InputWarning_H => #Sys.Alm_In_H,
            InputWarning_L => #Sys.Alm_In_L,
            State => #Sys.State,
            Error => #CMD.Alarm,
            ErrorBits => #Sys.Error_code);
   END_IF;
END_REGION

REGION Network 17: Обратное масштабирование в ручном режиме
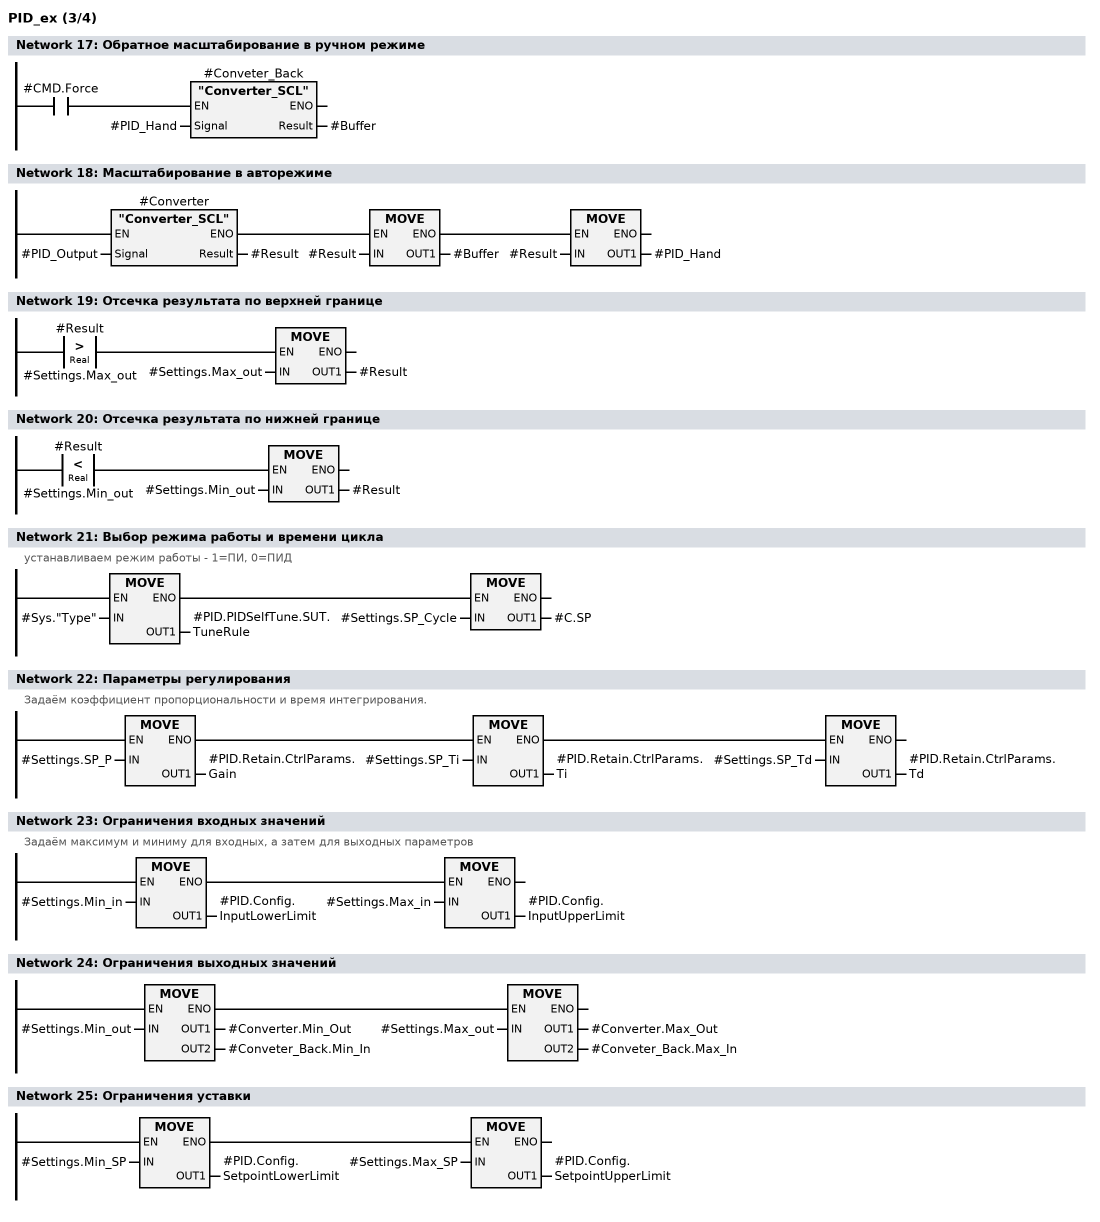
   RUNG wire#powerrail
      Contact( #CMD.Force )
      #Conveter_Back(Signal := #PID_Hand, Result => #Buffer)
   END_RUNG
   // the same network as SCL:
   IF #CMD.Force THEN
       #Conveter_Back(Signal := #PID_Hand, Result => #Buffer);   // "Converter_SCL"
   END_IF;
END_REGION

REGION Network 18: Масштабирование в авторежиме
   RUNG wire#powerrail
      #Converter(Signal := #PID_Output, Result => #Result)
      { S7_GenerateENO := "TRUE" } Move(in := #Result, out1 => #Buffer)
      { S7_GenerateENO := "TRUE" } Move(in := #Result, out1 => #PID_Hand)
   END_RUNG
   // the same network as SCL:
   // ENO of a box is taken as its EN; it also drops when the box reports an error
   #Converter(Signal := #PID_Output, Result => #Result, ENO => #_w1);   // "Converter_SCL"
   IF #_w1 THEN
       #Buffer := #Result;
       #PID_Hand := #Result;
   END_IF;
END_REGION

REGION Network 19: Отсечка результата по верхней границе
   RUNG wire#powerrail
      { S7_Templates := "SrcType := Real" } GT_Contact(in1 := #Result, in2 := #Settings.Max_out)
      Move(in := #Settings.Max_out, out1 => #Result)
   END_RUNG
   // the same network as SCL:
   IF #Result > #Settings.Max_out THEN #Result := #Settings.Max_out; END_IF;
END_REGION

REGION Network 20: Отсечка результата по нижней границе
   RUNG wire#powerrail
      { S7_Templates := "SrcType := Real" } LT_Contact(in1 := #Result, in2 := #Settings.Min_out)
      Move(in := #Settings.Min_out, out1 => #Result)
   END_RUNG
   // the same network as SCL:
   IF #Result < #Settings.Min_out THEN #Result := #Settings.Min_out; END_IF;
END_REGION

REGION Network 21: Выбор режима работы и времени цикла
   // устанавливаем режим работы - 1=ПИ, 0=ПИД
   RUNG wire#powerrail
      { S7_GenerateENO := "TRUE" } Move(in := #Sys."Type", out1 => #PID.PIDSelfTune.SUT.TuneRule)
      { S7_GenerateENO := "TRUE" } Move(in := #Settings.SP_Cycle, out1 => #C.SP)
   END_RUNG
   // the same network as SCL:
   // ENO of a box is taken as its EN; it also drops when the box reports an error
   #PID.PIDSelfTune.SUT.TuneRule := #Sys."Type";
   #C.SP := #Settings.SP_Cycle;
END_REGION

REGION Network 22: Параметры регулирования
   // Задаём коэффициент пропорциональности и время интегрирования.
   RUNG wire#powerrail
      { S7_GenerateENO := "TRUE" } Move(in := #Settings.SP_P, out1 => #PID.Retain.CtrlParams.Gain)
      { S7_GenerateENO := "TRUE" } Move(in := #Settings.SP_Ti, out1 => #PID.Retain.CtrlParams.Ti)
      { S7_GenerateENO := "TRUE" } Move(in := #Settings.SP_Td, out1 => #PID.Retain.CtrlParams.Td)
   END_RUNG
   // the same network as SCL:
   // ENO of a box is taken as its EN; it also drops when the box reports an error
   #PID.Retain.CtrlParams.Gain := #Settings.SP_P;
   #PID.Retain.CtrlParams.Ti := #Settings.SP_Ti;
   #PID.Retain.CtrlParams.Td := #Settings.SP_Td;
END_REGION

REGION Network 23: Ограничения входных значений
   // Задаём максимум и миниму для входных, а затем для выходных параметров
   RUNG wire#powerrail
      { S7_GenerateENO := "TRUE" } Move(in := #Settings.Min_in, out1 => #PID.Config.InputLowerLimit)
      { S7_GenerateENO := "TRUE" } Move(in := #Settings.Max_in, out1 => #PID.Config.InputUpperLimit)
   END_RUNG
   // the same network as SCL:
   // ENO of a box is taken as its EN; it also drops when the box reports an error
   #PID.Config.InputLowerLimit := #Settings.Min_in;
   #PID.Config.InputUpperLimit := #Settings.Max_in;
END_REGION

REGION Network 24: Ограничения выходных значений
   RUNG wire#powerrail
      { S7_GenerateENO := "TRUE" } Move(in := #Settings.Min_out, out1 => #Converter.Min_Out, out2 => #Conveter_Back.Min_In)
      { S7_GenerateENO := "TRUE" } Move(in := #Settings.Max_out, out1 => #Converter.Max_Out, out2 => #Conveter_Back.Max_In)
   END_RUNG
   // the same network as SCL:
   // ENO of a box is taken as its EN; it also drops when the box reports an error
   #Converter.Min_Out := #Settings.Min_out;
   #Conveter_Back.Min_In := #Settings.Min_out;
   #Converter.Max_Out := #Settings.Max_out;
   #Conveter_Back.Max_In := #Settings.Max_out;
END_REGION

REGION Network 25: Ограничения уставки
   RUNG wire#powerrail
      { S7_GenerateENO := "TRUE" } Move(in := #Settings.Min_SP, out1 => #PID.Config.SetpointLowerLimit)
      { S7_GenerateENO := "TRUE" } Move(in := #Settings.Max_SP, out1 => #PID.Config.SetpointUpperLimit)
   END_RUNG
   // the same network as SCL:
   // ENO of a box is taken as its EN; it also drops when the box reports an error
   #PID.Config.SetpointLowerLimit := #Settings.Min_SP;
   #PID.Config.SetpointUpperLimit := #Settings.Max_SP;
END_REGION

REGION Network 26: Сброс сброса
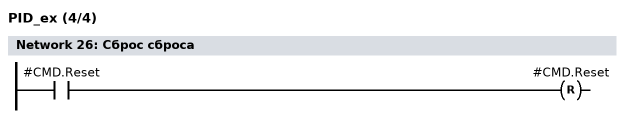
   RUNG wire#powerrail
      Contact( #CMD.Reset )
      R_Coil( #CMD.Reset )
   END_RUNG
   // the same network as SCL:
   IF #CMD.Reset THEN #CMD.Reset := FALSE; END_IF;
END_REGION
END_FUNCTION_BLOCK

ORGANIZATION_BLOCK "Diagnostic error interrupt"   // OB82, LAD, DiagnosticErrorInterrupt
{ S7_Optimized_Access := 'TRUE' }
VERSION : 0.1
// stored: IsIECCheckEnabled false, SetENOAutomatically false
   VAR_INPUT
      IO_State : Word;   // IO state of the HW object
      LADDR : HW_ANY;   // Hardware identifier
      Channel : UInt;   // Channel number
      MultiError : Bool;   // =true if more than one error is present
   END_VAR
BEGIN
END_ORGANIZATION_BLOCK

ORGANIZATION_BLOCK "Pull or plug of modules"   // OB83, LAD, PullOrPlugOfModules
{ S7_Optimized_Access := 'TRUE' }
VERSION : 0.1
// stored: IsIECCheckEnabled false, SetENOAutomatically false
   VAR_INPUT
      LADDR : HW_IO;   // Hardware identifier
      Event_Class : Byte;   // 16#38/39: module inserted, removed
      Fault_ID : Byte;   // Fault identifier
   END_VAR
BEGIN
END_ORGANIZATION_BLOCK

ORGANIZATION_BLOCK "Rack or station failure"   // OB86, LAD, RackOrStationFailure
{ S7_Optimized_Access := 'TRUE' }
VERSION : 0.1
// stored: IsIECCheckEnabled false, SetENOAutomatically false
   VAR_INPUT
      LADDR : HW_DEVICE;   // Hardware identifier
      Event_Class : Byte;   // Event class
      Fault_ID : Byte;   // Fault identifier
   END_VAR
BEGIN
END_ORGANIZATION_BLOCK

FUNCTION_BLOCK "Main_Logick"   // FB1, LAD
{ S7_Optimized_Access := 'FALSE' }
VERSION : 0.1
// stored: AutoNumber true, IsIECCheckEnabled false, SetENOAutomatically false, UDAEnableTagReadback false
   VAR DB_SPECIFIC
      Start : Bool;   // Запуск установки
      Start_Local : Bool;
      REQ_Pump : Bool;   // Запрос запуска насоса
      ev : Bool;
      Ready : Bool;   // Установка готова к работе
      Local : Bool;   // 0-местный, 1-дистанционный
      Mode : Bool;   // 0 - Работа по Гц, 1 - Работа по RM
      SP_Pump { S7_SetPoint := 'True'} : Real;   // уставка для работы по Гц
      RM : Real;   // Расходомер (получаем по MoodBus)
      RM_SP { S7_SetPoint := 'True'} : Real;   // Уставка расхода для насоса
      Level_Norm { S7_SetPoint := 'True'} : Real := 50.0;   // Рабочая точка насоса по уровню
      Distance { S7_SetPoint := 'True'} : Real := 500.0;   // Расстояние от ЩКД1 до скважины
      LE_Bar : Real;   // Показания датчика уровня на панели
      LE_Skvaz { S7_SetPoint := 'True'} : Real := 100.0;   // Глубина скважины
      LE_Skvaz_RCHV { S7_SetPoint := 'True'} : Real;   // Высота скважины относительно резервуара (для рассчета эфективности)
      Effect : Real;   // Эфективность скважины
      Alarm : Word;   // Слово аварий
      Alarms : Struct   // Список аварий
         Leak : Bool;   // Протечка
         Level_Norm : Bool;   // Уровень не в норме
         LE_Warning : Bool;   // Уровень ниже рабочей точки (Предупреждение)
         LE_Alarm : Bool;   // Уровень в аварийной зоне
      END_STRUCT;
   END_VAR
   VAR
      PID_Pump { S7_SetPoint := 'True'} : "PID_ex";   // ПИД Насоса
   END_VAR
   VAR_TEMP   // added for the SCL form of the ladder/FBD networks
      _w1 : Bool;
      _w2 : Bool;
      _w3 : Bool;
      _w4 : Bool;
   END_VAR
BEGIN

REGION Network 1: Готовность скважины к работе
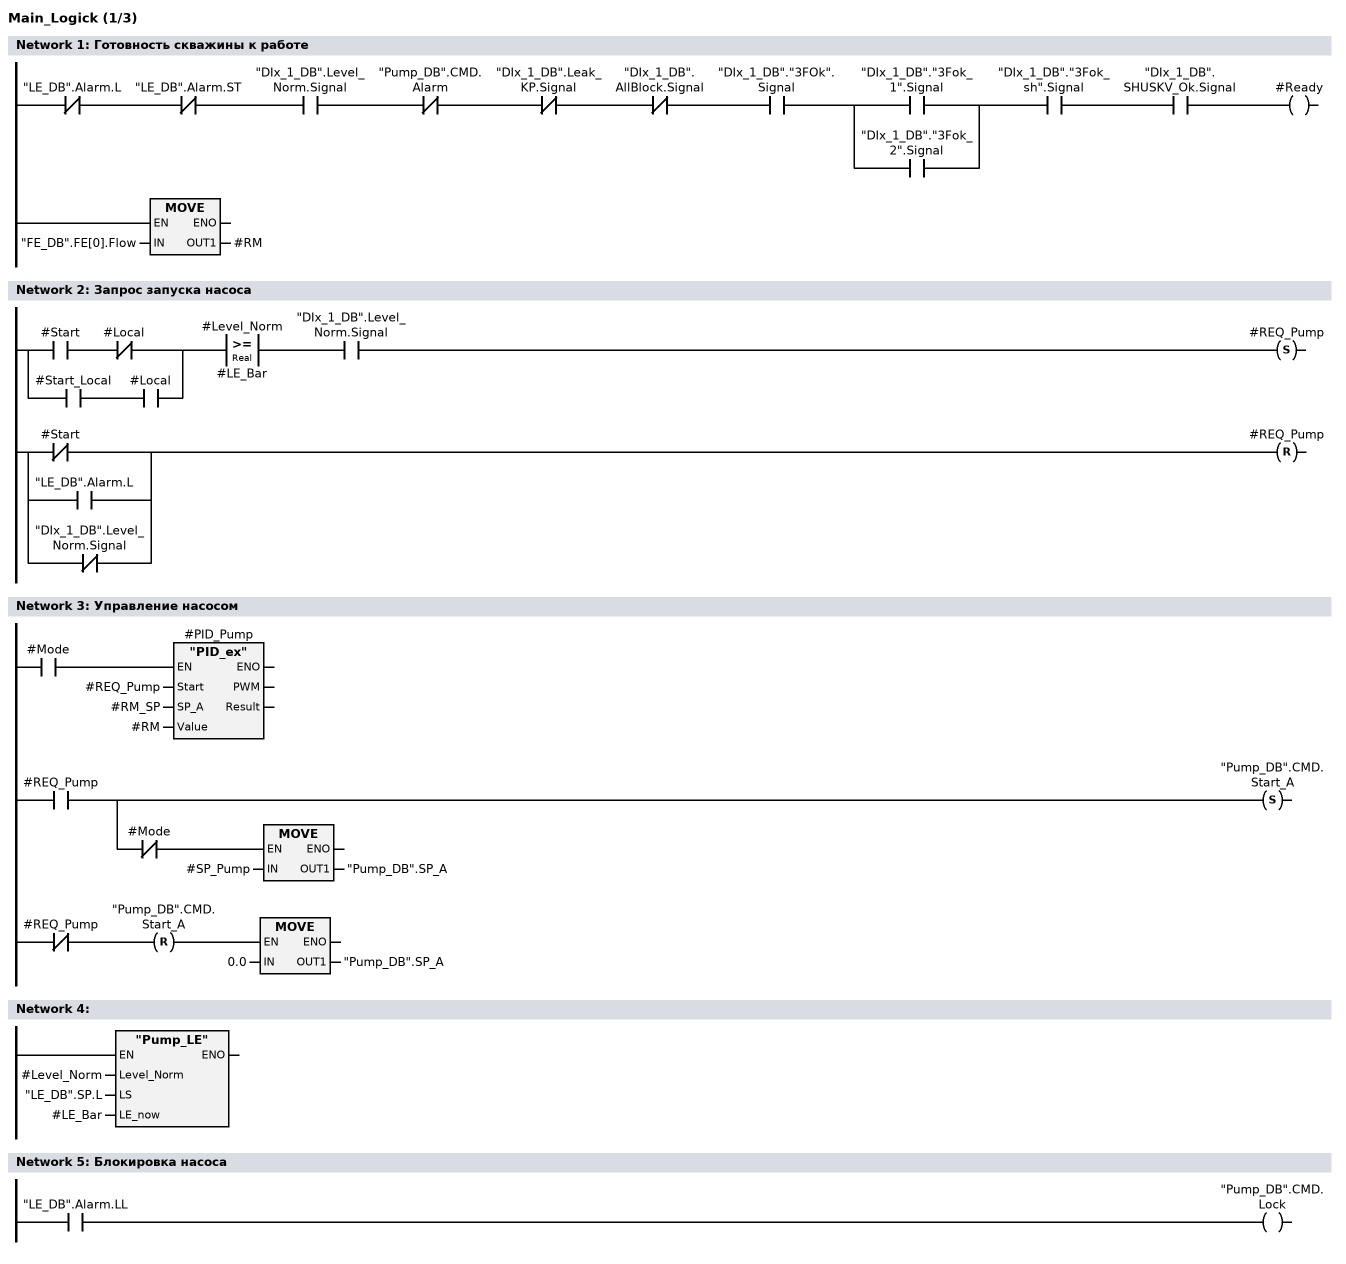
   RUNG wire#powerrail
      I_Contact( "LE_DB".Alarm.L )
      I_Contact( "LE_DB".Alarm.ST )
      Contact( "DIx_1_DB".Level_Norm.Signal )
      I_Contact( "Pump_DB".CMD.Alarm )
      I_Contact( "DIx_1_DB".Leak_KP.Signal )
      I_Contact( "DIx_1_DB".AllBlock.Signal )
      Contact( "DIx_1_DB"."3FOk".Signal )
      wire#w1
      Contact( "DIx_1_DB"."3Fok_1".Signal )
      wire#w2
      Contact( "DIx_1_DB"."3Fok_sh".Signal )
      Contact( "DIx_1_DB".SHUSKV_Ok.Signal )
      Coil( #Ready )
   END_RUNG
   RUNG wire#w1
      Contact( "DIx_1_DB"."3Fok_2".Signal )
   END_RUNG wire#w2
   RUNG wire#powerrail
      Move(in := "FE_DB".FE[0].Flow, out1 => #RM)
   END_RUNG
   // the same network as SCL:
   #Ready := NOT "LE_DB".Alarm.L AND NOT "LE_DB".Alarm.ST AND "DIx_1_DB".Level_Norm.Signal AND NOT "Pump_DB".CMD.Alarm AND NOT "DIx_1_DB".Leak_KP.Signal AND NOT "DIx_1_DB".AllBlock.Signal AND "DIx_1_DB"."3FOk".Signal AND ("DIx_1_DB"."3Fok_1".Signal OR "DIx_1_DB"."3Fok_2".Signal) AND "DIx_1_DB"."3Fok_sh".Signal AND "DIx_1_DB".SHUSKV_Ok.Signal;
   #RM := "FE_DB".FE[0].Flow;
END_REGION

REGION Network 2: Запрос запуска насоса
   RUNG wire#powerrail
      Contact( #Start )
      I_Contact( #Local )
      wire#w1
      { S7_Templates := "SrcType := Real" } GE_Contact(in1 := #Level_Norm, in2 := #LE_Bar)
      Contact( "DIx_1_DB".Level_Norm.Signal )
      S_Coil( #REQ_Pump )
   END_RUNG
   RUNG wire#powerrail
      Contact( #Start_Local )
      Contact( #Local )
   END_RUNG wire#w1
   RUNG wire#powerrail
      I_Contact( #Start )
      wire#w2
      R_Coil( #REQ_Pump )
   END_RUNG
   RUNG wire#powerrail
      Contact( "LE_DB".Alarm.L )
   END_RUNG wire#w2
   RUNG wire#powerrail
      I_Contact( "DIx_1_DB".Level_Norm.Signal )
   END_RUNG wire#w2
   // the same network as SCL:
   IF ((#Start AND NOT #Local) OR (#Start_Local AND #Local)) AND (#Level_Norm >= #LE_Bar) AND "DIx_1_DB".Level_Norm.Signal THEN
       #REQ_Pump := TRUE;
   END_IF;
   IF NOT #Start OR "LE_DB".Alarm.L OR NOT "DIx_1_DB".Level_Norm.Signal THEN #REQ_Pump := FALSE; END_IF;
END_REGION

REGION Network 3: Управление насосом
   RUNG wire#powerrail
      Contact( #Mode )
      #PID_Pump(Start := #REQ_Pump, SP_A := #RM_SP, Value := #RM, PWM =>, Result =>)
   END_RUNG
   RUNG wire#powerrail
      Contact( #REQ_Pump )
      wire#w1
      S_Coil( "Pump_DB".CMD.Start_A )
   END_RUNG
   RUNG wire#w1
      I_Contact( #Mode )
      Move(in := #SP_Pump, out1 => "Pump_DB".SP_A)
   END_RUNG
   RUNG wire#powerrail
      I_Contact( #REQ_Pump )
      R_Coil( "Pump_DB".CMD.Start_A )
      Move(in := 0.0, out1 => "Pump_DB".SP_A)
   END_RUNG
   // the same network as SCL:
   IF #Mode THEN
       #PID_Pump(Start := #REQ_Pump, SP_A := #RM_SP, Value := #RM);   // "PID_ex"
   END_IF;
   IF #REQ_Pump THEN "Pump_DB".CMD.Start_A := TRUE; END_IF;
   IF #REQ_Pump AND NOT #Mode THEN "Pump_DB".SP_A := #SP_Pump; END_IF;
   IF NOT #REQ_Pump THEN
       "Pump_DB".CMD.Start_A := FALSE;
       "Pump_DB".SP_A := 0.0;
   END_IF;
END_REGION

REGION Network 4
   RUNG wire#powerrail
      "Pump_LE"(Level_Norm := #Level_Norm, LS := "LE_DB".SP.L, LE_now := #LE_Bar)
   END_RUNG
   // the same network as SCL:
   "Pump_LE"(Level_Norm := #Level_Norm, LS := "LE_DB".SP.L, LE_now := #LE_Bar);
END_REGION

REGION Network 5: Блокировка насоса
   RUNG wire#powerrail
      Contact( "LE_DB".Alarm.LL )
      Coil( "Pump_DB".CMD.Lock )
   END_RUNG
   // the same network as SCL:
   "Pump_DB".CMD.Lock := "LE_DB".Alarm.LL;
END_REGION

REGION Network 6: Датчики перелива и уровня (Аварии)
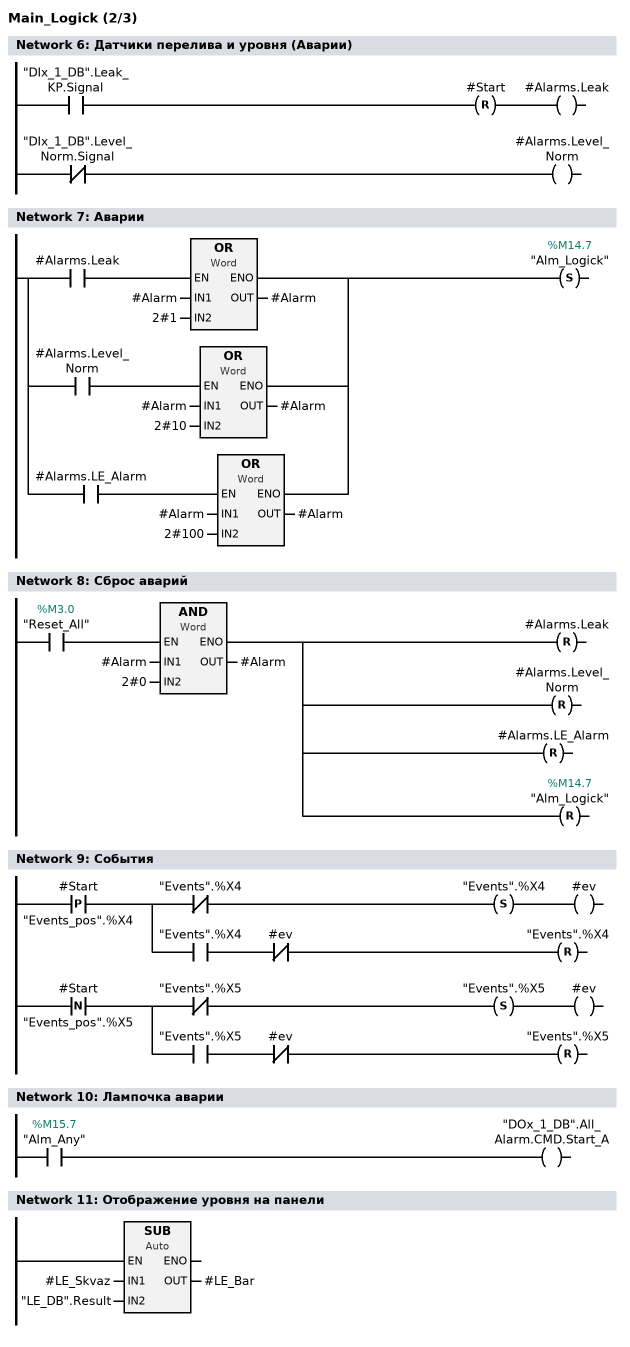
   RUNG wire#powerrail
      Contact( "DIx_1_DB".Leak_KP.Signal )
      R_Coil( #Start )
      Coil( #Alarms.Leak )
   END_RUNG
   RUNG wire#powerrail
      I_Contact( "DIx_1_DB".Level_Norm.Signal )
      Coil( #Alarms.Level_Norm )
   END_RUNG
   // the same network as SCL:
   IF "DIx_1_DB".Leak_KP.Signal THEN #Start := FALSE; END_IF;
   #Alarms.Leak := "DIx_1_DB".Leak_KP.Signal;
   #Alarms.Level_Norm := NOT "DIx_1_DB".Level_Norm.Signal;
END_REGION

REGION Network 7: Аварии
   IF #Alarms.Leak THEN #Alarm := #Alarm OR 2#1; END_IF;
   IF #Alarms.Level_Norm THEN #Alarm := #Alarm OR 2#10; END_IF;
   IF #Alarms.LE_Alarm THEN #Alarm := #Alarm OR 2#100; END_IF;
   IF #Alarms.Leak OR #Alarms.Level_Norm OR #Alarms.LE_Alarm THEN "Alm_Logick" := TRUE; END_IF;
END_REGION

REGION Network 8: Сброс аварий
   RUNG wire#powerrail
      Contact( "Reset_All" )
      { S7_Templates := "SrcType := Word"; S7_GenerateENO := "TRUE" } And(in1 := #Alarm, in2 := 2#0, out => #Alarm)
      wire#w1
      R_Coil( #Alarms.Leak )
   END_RUNG
   RUNG wire#w1
      R_Coil( #Alarms.Level_Norm )
   END_RUNG
   RUNG wire#w1
      R_Coil( #Alarms.LE_Alarm )
   END_RUNG
   RUNG wire#w1
      R_Coil( "Alm_Logick" )
   END_RUNG
   // the same network as SCL:
   IF "Reset_All" THEN
       #Alarm := #Alarm AND 2#0;
       #Alarms.Leak := FALSE;
       #Alarms.Level_Norm := FALSE;
       #Alarms.LE_Alarm := FALSE;
       "Alm_Logick" := FALSE;
   END_IF;
END_REGION

REGION Network 9: События
   RUNG wire#powerrail
      P_Contact(operand := #Start, bit := "Events_pos".%X4)
      wire#w1
      I_Contact( "Events".%X4 )
      S_Coil( "Events".%X4 )
      Coil( #ev )
   END_RUNG
   RUNG wire#w1
      Contact( "Events".%X4 )
      I_Contact( #ev )
      R_Coil( "Events".%X4 )
   END_RUNG
   RUNG wire#powerrail
      N_Contact(operand := #Start, bit := "Events_pos".%X5)
      wire#w2
      I_Contact( "Events".%X5 )
      S_Coil( "Events".%X5 )
      Coil( #ev )
   END_RUNG
   RUNG wire#w2
      Contact( "Events".%X5 )
      I_Contact( #ev )
      R_Coil( "Events".%X5 )
   END_RUNG
   // the same network as SCL:
   #_w1 := #Start AND NOT "Events_pos".%X4;   // rising edge of #Start
   "Events_pos".%X4 := #Start;
   #_w2 := #_w1 AND NOT "Events".%X4;
   IF #_w2 THEN "Events".%X4 := TRUE; END_IF;
   #ev := #_w2;
   IF #_w1 AND "Events".%X4 AND NOT #ev THEN "Events".%X4 := FALSE; END_IF;
   #_w3 := NOT #Start AND "Events_pos".%X5;   // falling edge of #Start
   "Events_pos".%X5 := #Start;
   #_w4 := #_w3 AND NOT "Events".%X5;
   IF #_w4 THEN "Events".%X5 := TRUE; END_IF;
   #ev := #_w4;
   IF #_w3 AND "Events".%X5 AND NOT #ev THEN "Events".%X5 := FALSE; END_IF;
END_REGION

REGION Network 10: Лампочка аварии
   RUNG wire#powerrail
      Contact( "Alm_Any" )
      Coil( "DOx_1_DB".All_Alarm.CMD.Start_A )
   END_RUNG
   // the same network as SCL:
   "DOx_1_DB".All_Alarm.CMD.Start_A := "Alm_Any";
END_REGION

REGION Network 11: Отображение уровня на панели
   RUNG wire#powerrail
      Sub(in1 := #LE_Skvaz, in2 := "LE_DB".Result, out => #LE_Bar)
   END_RUNG
   // the same network as SCL:
   #LE_Bar := #LE_Skvaz - "LE_DB".Result;
END_REGION

REGION Network 12: Рассчет эффективности скважины
